KUKA KRL program: MyProgram_341().src

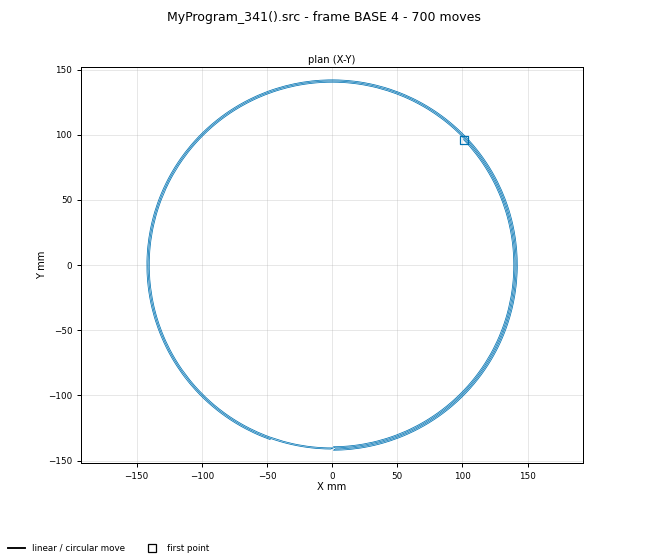
[picture p0: tool path of MyProgram_341().src in frame BASE 4, 700 of 700 moves have a stored position in this frame; points joined in program order, loops and branches not executed]
&ACCESS RVP
&REL 1
&PARAM TEMPLATE = C:\KRC\Roboter\Template\vorgabe
&PARAM EDITMASK = *
DEF MyProgram_341()
; ---- Setting reference (Base) ----
$BASE = BASE_DATA[4]

; --------------------------
; ---- Setting tool (TCP) ----
$TOOL = TOOL_DATA[3]
; --------------------------

$VEL.CP = VEL_APROX_PRINT
Startdeposition()
$VEL.CP = VEL_PRINT
LIN {X 100.8445,Y 96.2185,Z 191,A 42.0975,B 0.9774,C -0.019,E1 1.0995,E2 412.4998} C_DIS
LIN {X 103.8086,Y 93.0127,Z 191,A 40.4177,B 0.9774,C -0.0155,E1 1.1026,E2 414.1663} C_DIS
LIN {X 106.2355,Y 90.231,Z 191,A 38.3434,B 0.9775,C -0.0094,E1 1.1065,E2 416.3061} C_DIS
LIN {X 110.6605,Y 84.7459,Z 191,A 36.5482,B 0.9775,C -0.0077,E1 1.1094,E2 417.9718} C_DIS
LIN {X 113.1672,Y 81.369,Z 191,A 34.9648,B 0.9775,C -0.0043,E1 1.1119,E2 419.5381} C_DIS
LIN {X 115.7129,Y 77.7063,Z 191,A 33.5143,B 0.9775,C -0.0016,E1 1.1142,E2 420.9429} C_DIS
LIN {X 117.8631,Y 74.4035,Z 191,A 31.9484,B 0.9775,C 0.0021,E1 1.1165,E2 422.5025} C_DIS
LIN {X 120.2559,Y 70.4708,Z 191,A 30.262,B 0.9775,C 0.0059,E1 1.1189,E2 424.1645} C_DIS
LIN {X 122.5255,Y 66.4472,Z 191,A 28.5444,B 0.9775,C 0.0098,E1 1.1212,E2 425.8605} C_DIS
LIN {X 124.3166,Y 63.0275,Z 191,A 27.3294,B 0.9775,C 0.012,E1 1.1227,E2 427.0302} C_DIS
LIN {X 125.8319,Y 59.9448,Z 191,A 26.0722,B 0.9775,C 0.0149,E1 1.1242,E2 428.2687} C_DIS
LIN {X 128.0883,Y 54.9597,Z 191,A 23.995,B 0.9774,C 0.02,E1 1.1266,E2 430.3255} C_DIS
LIN {X 129.697,Y 51.0498,Z 191,A 22.4291,B 0.9774,C 0.0237,E1 1.1282,E2 431.8706} C_DIS
LIN {X 130.9681,Y 47.693,Z 191,A 21.1977,B 0.9772,C 0.0264,E1 1.1294,E2 433.0721} C_DIS
LIN {X 132.2016,Y 44.1567,Z 191,A 19.8499,B 0.9772,C 0.0295,E1 1.1306,E2 434.3965} C_DIS
LIN {X 133.196,Y 41.0607,Z 191,A 18.7703,B 0.9771,C 0.0318,E1 1.1314,E2 435.4443} C_DIS
LIN {X 134.1502,Y 37.8272,Z 191,A 17.3189,B 0.9769,C 0.0359,E1 1.1326,E2 436.9045} C_DIS
LIN {X 135.4414,Y 32.9058,Z 191,A 15.6224,B 0.9768,C 0.0396,E1 1.1337,E2 438.552} C_DIS
LIN {X 136.2147,Y 29.541,Z 191,A 14.3967,B 0.9767,C 0.0425,E1 1.1344,E2 439.7537} C_DIS
LIN {X 136.8872,Y 26.249,Z 191,A 12.5903,B 0.9764,C 0.0485,E1 1.1354,E2 441.6147} C_DIS
LIN {X 137.8072,Y 20.8924,Z 191,A 11.137,B 0.9763,C 0.0506,E1 1.136,E2 442.9697} C_DIS
LIN {X 138.3728,Y 16.7382,Z 191,A 9.6483,B 0.9761,C 0.0541,E1 1.1365,E2 444.4291} C_DIS
LIN {X 138.8051,Y 12.6771,Z 191,A 8.2382,B 0.9759,C 0.0574,E1 1.1369,E2 445.8054} C_DIS
LIN {X 139.1203,Y 8.5272,Z 191,A 6.7214,B 0.9757,C 0.0611,E1 1.1372,E2 447.2978} C_DIS
LIN {X 139.3137,Y 4.3756,Z 191,A 5.1532,B 0.9754,C 0.0651,E1 1.1374,E2 448.8488} C_DIS
LIN {X 139.3836,Y 0.2246,Z 191,A 3.614,B 0.9752,C 0.069,E1 1.1374,E2 450.3672} C_DIS
LIN {X 139.3302,Y -3.7808,Z 191,A 2.2878,B 0.9749,C 0.0719,E1 1.1374,E2 451.6522} C_DIS
LIN {X 139.1564,Y -7.9417,Z 191,A 0.7291,B 0.9746,C 0.0758,E1 1.1371,E2 453.1919} C_DIS
LIN {X 138.8913,Y -11.6781,Z 191,A -0.5528,B 0.9744,C 0.0787,E1 1.1368,E2 454.4406} C_DIS
LIN {X 138.519,Y -15.4917,Z 191,A -2.0184,B 0.9741,C 0.0825,E1 1.1364,E2 455.8927} C_DIS
LIN {X 138.008,Y -19.5189,Z 191,A -3.3769,B 0.9738,C 0.0855,E1 1.1359,E2 457.2109} C_DIS
LIN {X 137.3215,Y -23.8827,Z 191,A -5.0767,B 0.9735,C 0.0899,E1 1.1352,E2 458.8964} C_DIS
LIN {X 135.348,Y -33.2922,Z 191,A -8.6245,B 0.9726,C 0.0986,E1 1.1331,E2 462.3925} C_DIS
LIN {X 134.1503,Y -37.8269,Z 191,A -10.132,B 0.9723,C 0.1016,E1 1.132,E2 463.8445} C_DIS
LIN {X 133.1919,Y -41.0742,Z 191,A -11.393,B 0.972,C 0.1046,E1 1.131,E2 465.0888} C_DIS
LIN {X 132.027,Y -44.681,Z 191,A -12.8025,B 0.9716,C 0.108,E1 1.1298,E2 466.4792} C_DIS
LIN {X 130.6228,Y -48.6293,Z 191,A -14.2703,B 0.9712,C 0.1113,E1 1.1284,E2 467.9133} C_DIS
LIN {X 129.3401,Y -51.9444,Z 191,A -15.4509,B 0.971,C 0.1136,E1 1.1273,E2 469.0566} C_DIS
LIN {X 128.1203,Y -54.8857,Z 191,A -16.7235,B 0.9706,C 0.1169,E1 1.1259,E2 470.3252} C_DIS
LIN {X 126.5632,Y -58.385,Z 191,A -18.3527,B 0.97,C 0.1213,E1 1.124,E2 471.963} C_DIS
LIN {X 125.0675,Y -61.5237,Z 191,A -19.3037,B 0.9699,C 0.1225,E1 1.1229,E2 472.8492} C_DIS
LIN {X 123.5214,Y -64.5721,Z 191,A -20.5873,B 0.9695,C 0.1254,E1 1.1213,E2 474.117} C_DIS
LIN {X 121.4342,Y -68.4204,Z 191,A -22.2474,B 0.969,C 0.1292,E1 1.119,E2 475.7592} C_DIS
LIN {X 117.5792,Y -74.8523,Z 191,A -25.0092,B 0.9682,C 0.1352,E1 1.1151,E2 478.4787} C_DIS
LIN {X 115.0876,Y -78.629,Z 191,A -26.6462,B 0.9677,C 0.1386,E1 1.1126,E2 480.0859} C_DIS
LIN {X 112.552,Y -82.2179,Z 191,A -28.2704,B 0.9672,C 0.142,E1 1.11,E2 481.686} C_DIS
LIN {X 109.8372,Y -85.8109,Z 191,A -29.9359,B 0.9667,C 0.1454,E1 1.1072,E2 483.3268} C_DIS
LIN {X 106.958,Y -89.3737,Z 191,A -31.6211,B 0.9662,C 0.1488,E1 1.1042,E2 484.9856} C_DIS
LIN {X 104.0833,Y -92.706,Z 191,A -33.2121,B 0.9657,C 0.1518,E1 1.1013,E2 486.5471} C_DIS
LIN {X 101.0542,Y -95.9991,Z 191,A -34.8822,B 0.9652,C 0.1551,E1 1.0982,E2 488.1947} C_DIS
LIN {X 97.8841,Y -99.2293,Z 191,A -36.565,B 0.9647,C 0.1582,E1 1.0949,E2 489.8537} C_DIS
LIN {X 94.7472,Y -102.2285,Z 191,A -38.1412,B 0.9642,C 0.161,E1 1.0917,E2 491.4017} C_DIS
LIN {X 91.3868,Y -105.2433,Z 191,A -39.8212,B 0.9637,C 0.164,E1 1.0882,E2 493.0579} C_DIS
LIN {X 87.9612,Y -108.1227,Z 191,A -41.4803,B 0.9632,C 0.1669,E1 1.0847,E2 494.6926} C_DIS
LIN {X 84.472,Y -110.87,Z 191,A -43.1407,B 0.9628,C 0.1697,E1 1.081,E2 496.3307} C_DIS
LIN {X 80.7896,Y -113.5815,Z 191,A -44.8575,B 0.9623,C 0.1725,E1 1.0772,E2 498.0255} C_DIS
LIN {X 77.1218,Y -116.1031,Z 191,A -46.5386,B 0.9618,C 0.1752,E1 1.0733,E2 499.6865} C_DIS
LIN {X 73.2603,Y -118.5779,Z 191,A -48.3012,B 0.9613,C 0.178,E1 1.0691,E2 501.4329} C_DIS
LIN {X 69.8608,Y -120.6112,Z 191,A -49.8943,B 0.9608,C 0.1806,E1 1.0653,E2 503.0221} C_DIS
LIN {X 65.5664,Y -122.9992,Z 191,A -51.6426,B 0.9604,C 0.1828,E1 1.061,E2 504.7325} C_DIS
LIN {X 62.4534,Y -124.6089,Z 191,A -52.8854,B 0.9601,C 0.1842,E1 1.058,E2 505.9477} C_DIS
LIN {X 59.6812,Y -125.9579,Z 191,A -54.3785,B 0.9595,C 0.1871,E1 1.0541,E2 507.4745} C_DIS
LIN {X 56.1986,Y -127.5514,Z 191,A -55.6,B 0.9594,C 0.188,E1 1.0511,E2 508.6458} C_DIS
LIN {X 52.2827,Y -129.2037,Z 191,A -57.1304,B 0.959,C 0.1896,E1 1.0472,E2 510.1459} C_DIS
LIN {X 49.3407,Y -130.3564,Z 191,A -58.3976,B 0.9587,C 0.1912,E1 1.0439,E2 511.4093} C_DIS
LIN {X 45.7816,Y -131.6477,Z 191,A -59.8421,B 0.9584,C 0.1928,E1 1.0401,E2 512.8386} C_DIS
LIN {X 41.2319,Y -133.1436,Z 191,A -61.6603,B 0.958,C 0.1947,E1 1.0352,E2 514.6361} C_DIS
LIN {X 37.7566,Y -134.17,Z 191,A -62.9003,B 0.9579,C 0.1955,E1 1.032,E2 515.8404} C_DIS
LIN {X 34.7406,Y -134.983,Z 191,A -64.2072,B 0.9575,C 0.197,E1 1.0284,E2 517.1516} C_DIS
LIN {X 31.2504,Y -135.8329,Z 191,A -65.6672,B 0.9572,C 0.1985,E1 1.0244,E2 518.6101} C_DIS
LIN {X 24.229,Y -137.2596,Z 191,A -68.5094,B 0.9567,C 0.2009,E1 1.0165,E2 521.4391} C_DIS
LIN {X 19.9228,Y -137.9502,Z 191,A -70.2698,B 0.9564,C 0.2023,E1 1.0116,E2 523.1958} C_DIS
LIN {X 15.9492,Y -138.4669,Z 191,A -71.9027,B 0.9562,C 0.2036,E1 1.007,E2 524.8277} C_DIS
LIN {X 12.1677,Y -138.8499,Z 191,A -73.3225,B 0.956,C 0.2042,E1 1.0031,E2 526.2274} C_DIS
LIN {X 8.3965,Y -139.1284,Z 191,A -74.8296,B 0.9559,C 0.205,E1 0.9989,E2 527.7284} C_DIS
LIN {X 4.4323,Y -139.3121,Z 191,A -76.4575,B 0.9557,C 0.2059,E1 0.9943,E2 529.3567} C_DIS
LIN {X 0.9891,Y -139.3743,Z 191,A -77.3358,B 0.9559,C 0.205,E1 0.992,E2 530.156} C_DIS
Enddeposition()
LIN {X 0.9891,Y -139.3743,Z 191,A -77.3359,B 0.9559,C 0.205,E1 0.992,E2 530.1562} C_DIS
Startdeposition()
$VEL.CP = VEL_PRINT
LIN {X 2.4288,Y -140.2594,Z 191,A -76.5258,B 0.9476,C 0.2041,E1 0.9859,E2 529.3391} C_DIS
LIN {X 6.4097,Y -140.1353,Z 191,A -74.8363,B 0.9478,C 0.203,E1 0.9907,E2 527.6393} C_DIS
LIN {X 10.5728,Y -139.8818,Z 191,A -73.3277,B 0.9479,C 0.2025,E1 0.9949,E2 526.159} C_DIS
LIN {X 13.5665,Y -139.6228,Z 191,A -72.0791,B 0.9481,C 0.2016,E1 0.9984,E2 524.9064} C_DIS
LIN {X 17.8568,Y -139.1395,Z 191,A -70.3527,B 0.9484,C 0.2003,E1 1.0033,E2 523.1845} C_DIS
LIN {X 21.4621,Y -138.6287,Z 191,A -68.9845,B 0.9486,C 0.1995,E1 1.0071,E2 521.8332} C_DIS
LIN {X 24.5478,Y -138.1157,Z 191,A -67.4888,B 0.949,C 0.1976,E1 1.0113,E2 520.304} C_DIS
LIN {X 27.7783,Y -137.5024,Z 191,A -66.1559,B 0.9492,C 0.1963,E1 1.015,E2 518.9718} C_DIS
LIN {X 31.2997,Y -136.7437,Z 191,A -65.0397,B 0.9492,C 0.1961,E1 1.0179,E2 517.9078} C_DIS
LIN {X 34.4904,Y -135.9739,Z 191,A -63.7984,B 0.9495,C 0.195,E1 1.0213,E2 516.6805} C_DIS
LIN {X 38.0281,Y -135.0274,Z 191,A -62.3767,B 0.9498,C 0.1936,E1 1.0251,E2 515.2687} C_DIS
LIN {X 43.6634,Y -133.3133,Z 191,A -60.1874,B 0.9502,C 0.1915,E1 1.031,E2 513.1102} C_DIS
LIN {X 46.3959,Y -132.3862,Z 191,A -59.034,B 0.9505,C 0.1901,E1 1.034,E2 511.9596} C_DIS
LIN {X 49.306,Y -131.3293,Z 191,A -57.8285,B 0.9508,C 0.1886,E1 1.0372,E2 510.762} C_DIS
LIN {X 52.5839,Y -130.0515,Z 191,A -56.476,B 0.9511,C 0.187,E1 1.0407,E2 509.421} C_DIS
LIN {X 55.9899,Y -128.6222,Z 191,A -54.2348,B 0.9521,C 0.1817,E1 1.0468,E2 507.0695} C_DIS
LIN {X 62.3622,Y -125.6563,Z 191,A -52.699,B 0.9519,C 0.1829,E1 1.0502,E2 505.7302} C_DIS
LIN {X 64.8781,Y -124.376,Z 191,A -50.8289,B 0.9528,C 0.178,E1 1.0551,E2 503.7532} C_DIS
LIN {X 69.4356,Y -121.8922,Z 191,A -49.6152,B 0.9528,C 0.1784,E1 1.0578,E2 502.672} C_DIS
LIN {X 72.0547,Y -120.3627,Z 191,A -48.2313,B 0.9533,C 0.1756,E1 1.0612,E2 501.2658} C_DIS
LIN {X 75.8829,Y -117.9867,Z 191,A -46.4993,B 0.9538,C 0.1728,E1 1.0653,E2 499.5484} C_DIS
LIN {X 79.5681,Y -115.5334,Z 191,A -44.87,B 0.9542,C 0.1703,E1 1.069,E2 497.944} C_DIS
LIN {X 83.324,Y -112.8549,Z 191,A -43.1765,B 0.9547,C 0.1676,E1 1.0728,E2 496.277} C_DIS
LIN {X 86.9126,Y -110.1149,Z 191,A -41.4764,B 0.9552,C 0.1647,E1 1.0766,E2 494.5965} C_DIS
LIN {X 90.1823,Y -107.453,Z 191,A -39.9215,B 0.9557,C 0.162,E1 1.0799,E2 493.0647} C_DIS
LIN {X 93.5979,Y -104.4913,Z 191,A -38.2596,B 0.9562,C 0.1591,E1 1.0833,E2 491.4283} C_DIS
LIN {X 97.0336,Y -101.3089,Z 191,A -36.5299,B 0.9567,C 0.1559,E1 1.0868,E2 489.7237} C_DIS
LIN {X 100.354,Y -98.0212,Z 191,A -34.8379,B 0.9572,C 0.1528,E1 1.0901,E2 488.0616} C_DIS
LIN {X 103.4196,Y -94.781,Z 191,A -33.1724,B 0.9577,C 0.1495,E1 1.0932,E2 486.4173} C_DIS
LIN {X 106.4882,Y -91.32,Z 191,A -31.4671,B 0.9582,C 0.1462,E1 1.0963,E2 484.7371} C_DIS
LIN {X 109.4817,Y -87.7094,Z 191,A -29.754,B 0.9588,C 0.1427,E1 1.0993,E2 483.0516} C_DIS
LIN {X 112.2376,Y -84.1541,Z 191,A -28.1375,B 0.9592,C 0.1395,E1 1.102,E2 481.4654} C_DIS
LIN {X 114.7766,Y -80.656,Z 191,A -26.5389,B 0.9597,C 0.1362,E1 1.1046,E2 479.8893} C_DIS
LIN {X 117.2996,Y -76.9406,Z 191,A -24.9364,B 0.9602,C 0.1329,E1 1.107,E2 478.3184} C_DIS
LIN {X 120.1916,Y -72.3397,Z 191,A -22.7561,B 0.9609,C 0.1276,E1 1.1102,E2 476.1421} C_DIS
LIN {X 121.982,Y -69.2782,Z 191,A -21.7324,B 0.9611,C 0.1262,E1 1.1116,E2 475.1776} C_DIS
LIN {X 123.3706,Y -66.7748,Z 191,A -20.607,B 0.9614,C 0.1234,E1 1.1131,E2 474.0575} C_DIS
LIN {X 125.2761,Y -63.1242,Z 191,A -19.0934,B 0.9619,C 0.12,E1 1.1149,E2 472.5664} C_DIS
LIN {X 127.8258,Y -57.7868,Z 191,A -17.1962,B 0.9623,C 0.1165,E1 1.1171,E2 470.7403} C_DIS
LIN {X 129.5247,Y -53.8686,Z 191,A -15.5699,B 0.9628,C 0.1125,E1 1.1189,E2 469.1292} C_DIS
LIN {X 130.7911,Y -50.7163,Z 191,A -14.2895,B 0.9631,C 0.1094,E1 1.1202,E2 467.8627} C_DIS
LIN {X 132.3941,Y -46.373,Z 191,A -12.3171,B 0.9637,C 0.1039,E1 1.122,E2 465.8777} C_DIS
LIN {X 133.6698,Y -42.5544,Z 191,A -11.2361,B 0.9639,C 0.1025,E1 1.1229,E2 464.8738} C_DIS
LIN {X 134.773,Y -38.9229,Z 191,A -9.7971,B 0.9643,C 0.0989,E1 1.124,E2 463.4492} C_DIS
LIN {X 136.6408,Y -31.7502,Z 191,A -7.3212,B 0.9648,C 0.0937,E1 1.1257,E2 461.0471} C_DIS
LIN {X 137.2829,Y -28.8532,Z 191,A -6.168,B 0.9651,C 0.0906,E1 1.1264,E2 459.9012} C_DIS
LIN {X 137.9304,Y -25.5795,Z 191,A -4.8144,B 0.9654,C 0.0869,E1 1.1271,E2 458.548} C_DIS
LIN {X 138.7105,Y -20.9335,Z 191,A -3.3224,B 0.9657,C 0.084,E1 1.1277,E2 457.1136} C_DIS
LIN {X 139.1128,Y -18.0608,Z 191,A -2.2563,B 0.9659,C 0.0813,E1 1.1281,E2 456.0628} C_DIS
LIN {X 139.5316,Y -14.483,Z 191,A -0.9051,B 0.9662,C 0.0779,E1 1.1285,E2 454.7269} C_DIS
LIN {X 139.9067,Y -10.2319,Z 191,A 0.5882,B 0.9665,C 0.0744,E1 1.1288,E2 453.2663} C_DIS
LIN {X 140.1401,Y -6.3129,Z 191,A 1.9488,B 0.9667,C 0.0712,E1 1.129,E2 451.9374} C_DIS
LIN {X 140.2396,Y -3.4171,Z 191,A 3.1048,B 0.9669,C 0.068,E1 1.1291,E2 450.7843} C_DIS
LIN {X 140.2798,Y 0.701,Z 191,A 4.5452,B 0.9672,C 0.0646,E1 1.1291,E2 449.3754} C_DIS
LIN {X 140.1875,Y 5.1167,Z 191,A 6.0969,B 0.9674,C 0.061,E1 1.1291,E2 447.8562} C_DIS
LIN {X 140.0016,Y 8.8416,Z 191,A 7.3737,B 0.9676,C 0.058,E1 1.1288,E2 446.6112} C_DIS
LIN {X 139.7754,Y 11.8919,Z 191,A 8.4772,B 0.9677,C 0.0553,E1 1.1286,E2 445.5262} C_DIS
LIN {X 139.4287,Y 15.4394,Z 191,A 9.7987,B 0.9679,C 0.052,E1 1.1282,E2 444.2217} C_DIS
LIN {X 138.9585,Y 19.2214,Z 191,A 11.2418,B 0.9681,C 0.0483,E1 1.1277,E2 442.7928} C_DIS
LIN {X 138.162,Y 24.2893,Z 191,A 13.2764,B 0.9684,C 0.0428,E1 1.1267,E2 440.7651} C_DIS
LIN {X 137.4641,Y 27.9666,Z 191,A 14.449,B 0.9684,C 0.0405,E1 1.1261,E2 439.6384} C_DIS
LIN {X 136.328,Y 33.0638,Z 191,A 16.1697,B 0.9686,C 0.0368,E1 1.125,E2 437.9702} C_DIS
LIN {X 134.7053,Y 39.1541,Z 191,A 18.2378,B 0.9688,C 0.0324,E1 1.1236,E2 435.9662} C_DIS
LIN {X 133.5293,Y 42.9941,Z 191,A 19.8571,B 0.9689,C 0.0281,E1 1.1222,E2 434.3489} C_DIS
LIN {X 132.4144,Y 46.3145,Z 191,A 21.1201,B 0.9689,C 0.0251,E1 1.1211,E2 433.1068} C_DIS
LIN {X 131.2205,Y 49.5964,Z 191,A 22.3533,B 0.9691,C 0.0223,E1 1.1199,E2 431.8977} C_DIS
LIN {X 129.9725,Y 52.7799,Z 191,A 23.5651,B 0.9691,C 0.0195,E1 1.1187,E2 430.7088} C_DIS
LIN {X 128.8122,Y 55.5506,Z 191,A 24.8376,B 0.9691,C 0.0161,E1 1.1173,E2 429.4301} C_DIS
LIN {X 126.793,Y 60.0185,Z 191,A 26.3297,B 0.9692,C 0.0134,E1 1.1156,E2 428.0017} C_DIS
LIN {X 124.8732,Y 63.9155,Z 191,A 28.0232,B 0.9692,C 0.0092,E1 1.1135,E2 426.3178} C_DIS
LIN {X 123.0071,Y 67.4414,Z 191,A 29.5422,B 0.9693,C 0.0056,E1 1.1115,E2 424.8122} C_DIS
LIN {X 120.7502,Y 71.4042,Z 191,A 31.1652,B 0.9693,C 0.0021,E1 1.1093,E2 423.2186} C_DIS
LIN {X 118.4379,Y 75.177,Z 191,A 33.1475,B 0.9693,C -0.0032,E1 1.1063,E2 421.2142} C_DIS
LIN {X 115.92,Y 79.0046,Z 191,A 34.5042,B 0.9693,C -0.0053,E1 1.1043,E2 419.9209} C_DIS
LIN {X 113.0722,Y 83.0281,Z 191,A 36.2138,B 0.9693,C -0.0087,E1 1.1015,E2 418.2482} C_DIS
LIN {X 110.078,Y 86.9578,Z 191,A 38.2225,B 0.9693,C -0.0134,E1 1.098,E2 416.2402} C_DIS
LIN {X 107.8514,Y 89.7059,Z 191,A 39.2586,B 0.9693,C -0.0149,E1 1.0963,E2 415.2538} C_DIS
LIN {X 105.0814,Y 92.9348,Z 191,A 40.865,B 0.9691,C -0.0182,E1 1.0934,E2 413.663} C_DIS
LIN {X 101.9188,Y 96.3928,Z 191,A 42.5668,B 0.9691,C -0.0215,E1 1.0902,E2 411.9867} C_DIS
LIN {X 98.7421,Y 99.6445,Z 191,A 44.3488,B 0.969,C -0.0253,E1 1.0866,E2 410.2135} C_DIS
LIN {X 93.6427,Y 104.4511,Z 191,A 46.6153,B 0.9689,C -0.0287,E1 1.0821,E2 408.0181} C_DIS
LIN {X 91.2896,Y 106.5144,Z 191,A 47.9945,B 0.9688,C -0.0318,E1 1.0792,E2 406.6268} C_DIS
LIN {X 87.7142,Y 109.4778,Z 191,A 49.6935,B 0.9687,C -0.0348,E1 1.0755,E2 404.9513} C_DIS
LIN {X 84.1709,Y 112.2249,Z 191,A 51.39,B 0.9686,C -0.0378,E1 1.0718,E2 403.2707} C_DIS
LIN {X 78.7346,Y 116.1028,Z 191,A 53.9921,B 0.9684,C -0.0424,E1 1.0658,E2 400.6835} C_DIS
LIN {X 74.2059,Y 119.0483,Z 191,A 55.875,B 0.9683,C -0.0451,E1 1.0614,E2 398.8387} C_DIS
LIN {X 70.7179,Y 121.1533,Z 191,A 57.4143,B 0.9682,C -0.0475,E1 1.0577,E2 397.314} C_DIS
LIN {X 66.6844,Y 123.4192,Z 191,A 59.1449,B 0.968,C -0.05,E1 1.0535,E2 395.6021} C_DIS
LIN {X 62.523,Y 125.5769,Z 191,A 60.8209,B 0.968,C -0.0522,E1 1.0493,E2 393.9539} C_DIS
LIN {X 58.5898,Y 127.4589,Z 191,A 62.4897,B 0.9678,C -0.0545,E1 1.0451,E2 392.2982} C_DIS
LIN {X 55.4025,Y 128.8762,Z 191,A 63.7787,B 0.9677,C -0.0561,E1 1.0418,E2 391.0251} C_DIS
LIN {X 51.8629,Y 130.3421,Z 191,A 65.2128,B 0.9676,C -0.0579,E1 1.0381,E2 389.6062} C_DIS
LIN {X 48.9366,Y 131.4676,Z 191,A 66.4229,B 0.9675,C -0.0594,E1 1.0349,E2 388.4044} C_DIS
LIN {X 45.7519,Y 132.6095,Z 191,A 67.7199,B 0.9675,C -0.0609,E1 1.0315,E2 387.1173} C_DIS
LIN {X 42.6175,Y 133.6496,Z 191,A 70.0962,B 0.9671,C -0.0659,E1 1.0248,E2 384.6231} C_DIS
LIN {X 34.6875,Y 135.9239,Z 191,A 71.9236,B 0.9671,C -0.0648,E1 1.0203,E2 382.9733} C_DIS
LIN {X 30.496,Y 136.9262,Z 191,A 74.095,B 0.9669,C -0.068,E1 1.0142,E2 380.7559} C_DIS
LIN {X 27.1654,Y 137.6271,Z 191,A 75.1328,B 0.9669,C -0.0683,E1 1.0114,E2 379.7584} C_DIS
LIN {X 24.2811,Y 138.1634,Z 191,A 76.3446,B 0.9669,C -0.0694,E1 1.008,E2 378.5453} C_DIS
LIN {X 19.9734,Y 138.8511,Z 191,A 78.0673,B 0.9667,C -0.0708,E1 1.0033,E2 376.8298} C_DIS
LIN {X 16.0453,Y 139.3608,Z 191,A 79.5373,B 0.9667,C -0.0716,E1 0.9992,E2 375.377} C_DIS
LIN {X 11.9143,Y 139.7735,Z 191,A 81.1822,B 0.9666,C -0.0727,E1 0.9946,E2 373.7383} C_DIS
LIN {X 8.3688,Y 140.0307,Z 191,A 82.5796,B 0.9666,C -0.0734,E1 0.9906,E2 372.3475} C_DIS
LIN {X 4.3944,Y 140.2124,Z 191,A 84.238,B 0.9665,C -0.0744,E1 0.9859,E2 370.686} C_DIS
LIN {X 0.4701,Y 140.28,Z 191,A 85.7526,B 0.9665,C -0.075,E1 0.9817,E2 369.1818} C_DIS
LIN {X -3.8447,Y 140.2277,Z 191,A 87.4841,B 0.9664,C -0.0756,E1 0.9768,E2 367.4543} C_DIS
LIN {X -8.1948,Y 140.0414,Z 191,A 89.2607,B 0.9664,C -0.0762,E1 0.9718,E2 365.6787} C_DIS
LIN {X -11.8972,Y 139.7749,Z 191,A 90.7411,B 0.9664,C -0.0765,E1 0.9676,E2 364.2029} C_DIS
LIN {X -16.0691,Y 139.3579,Z 191,A 92.4601,B 0.9663,C -0.0767,E1 0.9628,E2 362.4839} C_DIS
LIN {X -20.8516,Y 138.7232,Z 191,A 94.5728,B 0.9663,C -0.0771,E1 0.9568,E2 360.3563} C_DIS
LIN {X -24.7655,Y 138.0768,Z 191,A 95.986,B 0.9663,C -0.0767,E1 0.9529,E2 358.9668} C_DIS
LIN {X -28.6695,Y 137.3211,Z 191,A 97.6024,B 0.9663,C -0.0765,E1 0.9484,E2 357.3521} C_DIS
LIN {X -32.3615,Y 136.4972,Z 191,A 99.0478,B 0.9663,C -0.0761,E1 0.9445,E2 355.9184} C_DIS
LIN {X -35.0189,Y 135.8398,Z 191,A 100.2628,B 0.9663,C -0.076,E1 0.9411,E2 354.6932} C_DIS
LIN {X -37.9053,Y 135.0618,Z 191,A 101.5938,B 0.9663,C -0.0758,E1 0.9375,E2 353.3506} C_DIS
LIN {X -41.2345,Y 134.0829,Z 191,A 103.0152,B 0.9663,C -0.0753,E1 0.9336,E2 351.9294} C_DIS
LIN {X -44.7517,Y 132.9509,Z 191,A 104.5488,B 0.9664,C -0.0746,E1 0.9295,E2 350.3939} C_DIS
LIN {X -48.4055,Y 131.6665,Z 191,A 106.1601,B 0.9665,C -0.0739,E1 0.9252,E2 348.7802} C_DIS
LIN {X -51.1258,Y 130.6319,Z 191,A 107.4182,B 0.9665,C -0.0732,E1 0.9218,E2 347.5149} C_DIS
LIN {X -56.4675,Y 128.4137,Z 191,A 109.9431,B 0.9667,C -0.0718,E1 0.9152,E2 344.9731} C_DIS
LIN {X -59.2165,Y 127.1691,Z 191,A 111.1417,B 0.9667,C -0.0708,E1 0.9122,E2 343.7789} C_DIS
LIN {X -62.702,Y 125.4886,Z 191,A 112.7735,B 0.9668,C -0.0696,E1 0.908,E2 342.1423} C_DIS
LIN {X -65.7052,Y 123.9417,Z 191,A 114.2628,B 0.9669,C -0.0684,E1 0.9042,E2 340.6415} C_DIS
LIN {X -70.5272,Y 121.2641,Z 191,A 116.7091,B 0.967,C -0.0663,E1 0.8982,E2 338.1747} C_DIS
LIN {X -74.6394,Y 118.7772,Z 191,A 118.7378,B 0.9672,C -0.0642,E1 0.8933,E2 336.1397} C_DIS
LIN {X -78.1585,Y 116.4918,Z 191,A 120.775,B 0.9673,C -0.0623,E1 0.8884,E2 334.0669} C_DIS
LIN {X -82.3299,Y 113.5816,Z 191,A 122.6839,B 0.9675,C -0.0596,E1 0.884,E2 332.1783} C_DIS
LIN {X -85.1351,Y 111.4945,Z 191,A 124.4137,B 0.9675,C -0.0578,E1 0.8801,E2 330.4151} C_DIS
LIN {X -88.798,Y 108.5997,Z 191,A 126.447,B 0.9678,C -0.0551,E1 0.8756,E2 328.3684} C_DIS
LIN {X -92.093,Y 105.8202,Z 191,A 128.4084,B 0.9679,C -0.0524,E1 0.8713,E2 326.385} C_DIS
LIN {X -95.4496,Y 102.8027,Z 191,A 130.4234,B 0.9681,C -0.0495,E1 0.8671,E2 324.3515} C_DIS
LIN {X -98.6352,Y 99.7507,Z 191,A 132.4213,B 0.9682,C -0.0465,E1 0.863,E2 322.332} C_DIS
LIN {X -101.8138,Y 96.5042,Z 191,A 134.4577,B 0.9684,C -0.0432,E1 0.859,E2 320.2757} C_DIS
LIN {X -104.8181,Y 93.2328,Z 191,A 136.4679,B 0.9685,C -0.0398,E1 0.8552,E2 318.2438} C_DIS
LIN {X -107.7692,Y 89.8052,Z 191,A 138.4956,B 0.9686,C -0.0362,E1 0.8515,E2 316.1961} C_DIS
LIN {X -110.5694,Y 86.3341,Z 191,A 140.6663,B 0.9688,C -0.0325,E1 0.8476,E2 313.9854} C_DIS
LIN {X -114.8976,Y 80.4844,Z 191,A 144.4492,B 0.969,C -0.026,E1 0.8413,E2 310.1078} C_DIS
LIN {X -117.6144,Y 76.4582,Z 191,A 146.1159,B 0.969,C -0.0219,E1 0.8387,E2 308.4803} C_DIS
LIN {X -121.8922,Y 69.4356,Z 191,A 149.6168,B 0.9692,C -0.0142,E1 0.8337,E2 304.9647} C_DIS
LIN {X -123.3498,Y 66.8131,Z 191,A 151.4066,B 0.9692,C -0.011,E1 0.8311,E2 303.1077} C_DIS
LIN {X -125.0943,Y 63.4813,Z 191,A 152.9992,B 0.9692,C -0.0073,E1 0.8291,E2 301.5092} C_DIS
LIN {X -127.4467,Y 58.6161,Z 191,A 155.444,B 0.9693,C -0.0018,E1 0.8261,E2 299.0369} C_DIS
LIN {X -129.9834,Y 52.753,Z 191,A 158.4922,B 0.9693,C 0.005,E1 0.8227,E2 295.9367} C_DIS
LIN {X -130.907,Y 50.4182,Z 191,A 159.7153,B 0.9693,C 0.0078,E1 0.8214,E2 294.6899} C_DIS
LIN {X -131.9573,Y 47.5997,Z 191,A 161.2886,B 0.9693,C 0.0112,E1 0.8199,E2 293.0746} C_DIS
LIN {X -133.199,Y 44.0068,Z 191,A 162.9736,B 0.9692,C 0.0153,E1 0.8184,E2 291.374} C_DIS
LIN {X -134.211,Y 40.816,Z 191,A 164.6066,B 0.9692,C 0.0191,E1 0.817,E2 289.7086} C_DIS
LIN {X -135.1979,Y 37.4185,Z 191,A 166.8546,B 0.969,C 0.0237,E1 0.8153,E2 287.3601} C_DIS
LIN {X -136.3308,Y 33.0521,Z 191,A 168.4865,B 0.969,C 0.0284,E1 0.8142,E2 285.7561} C_DIS
LIN {X -137.0064,Y 30.1337,Z 191,A 169.9402,B 0.9688,C 0.0319,E1 0.8133,E2 284.274} C_DIS
LIN {X -137.8444,Y 26.0295,Z 191,A 171.8674,B 0.9686,C 0.0368,E1 0.8122,E2 282.3202} C_DIS
LIN {X -139.0055,Y 18.8799,Z 191,A 175.8108,B 0.9682,C 0.0459,E1 0.8105,E2 278.2514} C_DIS
LIN {X -139.4832,Y 14.9325,Z 191,A 177.2484,B 0.968,C 0.0502,E1 0.8101,E2 276.839} C_DIS
LIN {X -139.8778,Y 10.6278,Z 191,A -179.6827,B 0.9677,C 0.0563,E1 0.8094,E2 273.6001} C_DIS
LIN {X -140.2195,Y 4.1391,Z 191,A -177.8678,B 0.9673,C 0.063,E1 0.8092,E2 271.8975} C_DIS
LIN {X -140.2443,Y -3.2474,Z 191,A -174.1217,B 0.9666,C 0.0721,E1 0.8092,E2 268.0572} C_DIS
LIN {X -139.8415,Y -11.1088,Z 191,A -170.0509,B 0.9659,C 0.0818,E1 0.8099,E2 263.874} C_DIS
LIN {X -139.2722,Y -16.7876,Z 191,A -167.5021,B 0.9653,C 0.0884,E1 0.8107,E2 261.2971} C_DIS
LIN {X -137.9392,Y -25.5336,Z 191,A -163.3295,B 0.9643,C 0.0988,E1 0.8126,E2 257.0506} C_DIS
LIN {X -137.3992,Y -28.2855,Z 191,A -161.9601,B 0.9639,C 0.102,E1 0.8133,E2 255.6511} C_DIS
LIN {X -136.7276,Y -31.3699,Z 191,A -160.4707,B 0.9635,C 0.1056,E1 0.8143,E2 254.1348} C_DIS
LIN {X -135.9581,Y -34.5525,Z 191,A -158.866,B 0.9631,C 0.1094,E1 0.8154,E2 252.4939} C_DIS
LIN {X -135.0462,Y -37.9609,Z 191,A -157.1666,B 0.9627,C 0.1134,E1 0.8166,E2 250.7594} C_DIS
LIN {X -134.0581,Y -41.3155,Z 191,A -155.5401,B 0.9622,C 0.1172,E1 0.818,E2 249.1061} C_DIS
LIN {X -132.6865,Y -45.5296,Z 191,A -152.9972,B 0.9616,C 0.1223,E1 0.8204,E2 246.4615} C_DIS
LIN {X -131.3592,Y -49.2262,Z 191,A -151.9914,B 0.9611,C 0.1261,E1 0.8213,E2 245.5401} C_DIS
LIN {X -130.6363,Y -51.1145,Z 191,A -150.635,B 0.9608,C 0.1284,E1 0.8227,E2 244.1098} C_DIS
LIN {X -128.913,Y -55.3174,Z 191,A -148.6681,B 0.9601,C 0.1331,E1 0.8248,E2 242.128} C_DIS
LIN {X -127.5583,Y -58.3749,Z 191,A -146.7657,B 0.9596,C 0.1366,E1 0.8271,E2 240.1503} C_DIS
LIN {X -125.7295,Y -62.2136,Z 191,A -145.0019,B 0.959,C 0.1408,E1 0.8293,E2 238.3832} C_DIS
LIN {X -124.3202,Y -64.9844,Z 191,A -143.5199,B 0.9586,C 0.1438,E1 0.8312,E2 236.8714} C_DIS
LIN {X -122.3736,Y -68.5838,Z 191,A -141.4833,B 0.958,C 0.1478,E1 0.834,E2 234.7832} C_DIS
LIN {X -120.1597,Y -72.3927,Z 191,A -139.3765,B 0.9574,C 0.1518,E1 0.8371,E2 232.6328} C_DIS
LIN {X -117.5681,Y -76.5295,Z 191,A -137.2553,B 0.9567,C 0.1562,E1 0.8403,E2 230.4938} C_DIS
LIN {X -115.1138,Y -80.1736,Z 191,A -135.1918,B 0.956,C 0.16,E1 0.8437,E2 228.3919} C_DIS
LIN {X -109.0235,Y -88.2776,Z 191,A -130.9065,B 0.9546,C 0.1683,E1 0.851,E2 224.0868} C_DIS
LIN {X -105.3142,Y -92.6716,Z 191,A -127.9292,B 0.9539,C 0.1725,E1 0.8566,E2 221.0184} C_DIS
LIN {X -102.2596,Y -96.0316,Z 191,A -125.8675,B 0.9533,C 0.1757,E1 0.8606,E2 218.9266} C_DIS
LIN {X -97.1105,Y -101.2354,Z 191,A -122.0719,B 0.9524,C 0.1802,E1 0.8685,E2 215.0126} C_DIS
LIN {X -93.4502,Y -104.6235,Z 191,A -120.0576,B 0.9518,C 0.1834,E1 0.8727,E2 213.0017} C_DIS
LIN {X -90.4494,Y -107.2288,Z 191,A -118.9223,B 0.9513,C 0.1862,E1 0.875,E2 211.9384} C_DIS
LIN {X -86.5162,Y -110.4263,Z 191,A -116.4374,B 0.9508,C 0.1888,E1 0.8806,E2 209.3923} C_DIS
LIN {X -82.1503,Y -113.7118,Z 191,A -114.075,B 0.9502,C 0.1916,E1 0.886,E2 207.0104} C_DIS
LIN {X -78.6984,Y -116.1273,Z 191,A -112.1661,B 0.9498,C 0.1934,E1 0.8905,E2 205.0735} C_DIS
LIN {X -75.1214,Y -118.473,Z 191,A -110.2949,B 0.9495,C 0.1953,E1 0.895,E2 203.1837} C_DIS
LIN {X -71.254,Y -120.8384,Z 191,A -108.3133,B 0.9491,C 0.197,E1 0.8998,E2 201.1824} C_DIS
LIN {X -67.1186,Y -123.1832,Z 191,A -106.1291,B 0.9488,C 0.1985,E1 0.9053,E2 198.9617} C_DIS
LIN {X -63.0139,Y -125.3322,Z 191,A -104.4884,B 0.9484,C 0.2005,E1 0.9093,E2 197.3582} C_DIS
LIN {X -60.216,Y -126.6986,Z 191,A -103.0657,B 0.9482,C 0.2013,E1 0.913,E2 195.9126} C_DIS
LIN {X -57.0526,Y -128.1542,Z 191,A -101.6196,B 0.948,C 0.2023,E1 0.9167,E2 194.4627} C_DIS
LIN {X -53.778,Y -129.5626,Z 191,A -100.1387,B 0.9478,C 0.2032,E1 0.9206,E2 192.9777} C_DIS
LIN {X -50.83,Y -130.7469,Z 191,A -98.752,B 0.9477,C 0.2038,E1 0.9243,E2 191.5772} C_DIS
LIN {X -47.4936,Y -131.9956,Z 191,A -97.257,B 0.9475,C 0.2045,E1 0.9283,E2 190.0758} C_DIS
LIN {X -37.0814,Y -135.2922,Z 191,A -92.7922,B 0.9471,C 0.2062,E1 0.9404,E2 185.6095} C_DIS
LIN {X -30.0812,Y -137.0177,Z 191,A -89.8663,B 0.9471,C 0.2068,E1 0.9484,E2 182.6853} C_DIS
LIN {X -26.3218,Y -137.7885,Z 191,A -88.1757,B 0.9471,C 0.2066,E1 0.9532,E2 180.9756} C_DIS
LIN {X -22.8732,Y -138.403,Z 191,A -86.7287,B 0.9471,C 0.2066,E1 0.9572,E2 179.5255} C_DIS
LIN {X -19.4647,Y -138.9238,Z 191,A -85.3227,B 0.9471,C 0.2065,E1 0.9611,E2 178.1193} C_DIS
LIN {X -15.7103,Y -139.3995,Z 191,A -83.6759,B 0.9471,C 0.206,E1 0.9658,E2 176.4566} C_DIS
LIN {X -11.1977,Y -139.834,Z 191,A -81.8256,B 0.9473,C 0.2056,E1 0.971,E2 174.6056} C_DIS
LIN {X -7.0178,Y -140.1047,Z 191,A -80.2259,B 0.9473,C 0.2054,E1 0.9755,E2 173.0218} C_DIS
LIN {X -3.4723,Y -140.238,Z 191,A -78.8632,B 0.9473,C 0.2051,E1 0.9793,E2 171.6713} C_DIS
LIN {X 0.9989,Y -140.2749,Z 191,A -77.1882,B 0.9475,C 0.2047,E1 0.984,E2 170.0179} C_DIS
Enddeposition()
LIN {X 0.9989,Y -140.2749,Z 191,A -77.1882,B 0.9475,C 0.2047,E1 0.984,E2 170.0179} C_DIS
Startdeposition()
$VEL.CP = VEL_PRINT
LIN {X -1.0513,Y -141.1757,Z 191,A -78.2711,B 0.9179,C 0.2049,E1 0.9515,E2 171.1715} C_DIS
LIN {X -5.3673,Y -141.0773,Z 191,A -79.9095,B 0.9179,C 0.2053,E1 0.9469,E2 172.7937} C_DIS
LIN {X -8.8162,Y -140.9038,Z 191,A -81.251,B 0.9178,C 0.2055,E1 0.9431,E2 174.1269} C_DIS
LIN {X -11.9765,Y -140.6703,Z 191,A -82.6035,B 0.9176,C 0.2061,E1 0.9393,E2 175.49} C_DIS
LIN {X -15.6835,Y -140.3065,Z 191,A -84.1899,B 0.9176,C 0.2065,E1 0.9348,E2 177.0884} C_DIS
LIN {X -19.9252,Y -139.766,Z 191,A -85.8094,B 0.9176,C 0.2065,E1 0.9303,E2 178.6912} C_DIS
LIN {X -23.2557,Y -139.2505,Z 191,A -87.1888,B 0.9176,C 0.2065,E1 0.9264,E2 180.073} C_DIS
LIN {X -26.8832,Y -138.5964,Z 191,A -88.6783,B 0.9176,C 0.2065,E1 0.9223,E2 181.5622} C_DIS
LIN {X -31.0404,Y -137.725,Z 191,A -90.8437,B 0.9174,C 0.2072,E1 0.9161,E2 183.7947} C_DIS
LIN {X -35.2441,Y -136.71,Z 191,A -92.1868,B 0.9177,C 0.206,E1 0.9126,E2 185.0766} C_DIS
LIN {X -39.285,Y -135.6036,Z 191,A -94.4882,B 0.9175,C 0.2067,E1 0.9061,E2 187.4688} C_DIS
LIN {X -44.1423,Y -134.1013,Z 191,A -96.1549,B 0.9179,C 0.2051,E1 0.9017,E2 189.0768} C_DIS
LIN {X -47.6713,Y -132.887,Z 191,A -97.5862,B 0.918,C 0.2043,E1 0.8979,E2 190.4959} C_DIS
LIN {X -51.201,Y -131.5672,Z 191,A -99.1565,B 0.9182,C 0.2035,E1 0.8938,E2 192.0729} C_DIS
LIN {X -54.692,Y -130.155,Z 191,A -100.7423,B 0.9184,C 0.2027,E1 0.8896,E2 193.6678} C_DIS
LIN {X -58.558,Y -128.464,Z 191,A -102.5916,B 0.9186,C 0.2017,E1 0.8848,E2 195.538} C_DIS
LIN {X -62.73,Y -126.4772,Z 191,A -104.491,B 0.9189,C 0.2003,E1 0.8799,E2 197.4413} C_DIS
LIN {X -67.6372,Y -123.9243,Z 191,A -106.9008,B 0.9193,C 0.1985,E1 0.8738,E2 199.8763} C_DIS
LIN {X -71.4441,Y -121.7693,Z 191,A -108.7794,B 0.9196,C 0.1969,E1 0.8692,E2 201.7706} C_DIS
LIN {X -75.3483,Y -119.3928,Z 191,A -110.7404,B 0.92,C 0.1951,E1 0.8644,E2 203.7477} C_DIS
LIN {X -79.286,Y -116.8151,Z 191,A -112.9014,B 0.9205,C 0.1931,E1 0.8593,E2 205.9461} C_DIS
LIN {X -85.4007,Y -112.423,Z 191,A -116.0931,B 0.9212,C 0.1893,E1 0.8519,E2 209.1583} C_DIS
LIN {X -89.0391,Y -109.5637,Z 191,A -118.1076,B 0.9217,C 0.1868,E1 0.8475,E2 211.193} C_DIS
LIN {X -93.133,Y -106.1057,Z 191,A -120.4873,B 0.9224,C 0.1838,E1 0.8423,E2 213.603} C_DIS
LIN {X -96.5044,Y -103.0488,Z 191,A -123.3072,B 0.9228,C 0.1814,E1 0.8362,E2 216.5654} C_DIS
LIN {X -101.0981,Y -98.5462,Z 191,A -125.0656,B 0.9238,C 0.1766,E1 0.833,E2 218.1991} C_DIS
LIN {X -104.341,Y -95.1055,Z 191,A -127.5123,B 0.9244,C 0.1734,E1 0.8281,E2 220.723} C_DIS
LIN {X -108.3032,Y -90.5675,Z 191,A -130.1894,B 0.9252,C 0.1689,E1 0.8231,E2 223.4336} C_DIS
LIN {X -114.419,Y -82.7063,Z 191,A -134.4476,B 0.9266,C 0.1609,E1 0.8158,E2 227.7227} C_DIS
LIN {X -116.1948,Y -80.1929,Z 191,A -136.1485,B 0.9271,C 0.1583,E1 0.8129,E2 229.4887} C_DIS
LIN {X -118.4424,Y -76.8336,Z 191,A -138.0895,B 0.9277,C 0.1548,E1 0.8099,E2 231.4727} C_DIS
LIN {X -121.0046,Y -72.7326,Z 191,A -140.2526,B 0.9284,C 0.1504,E1 0.8066,E2 233.664} C_DIS
LIN {X -123.2553,Y -68.8497,Z 191,A -142.288,B 0.9291,C 0.1462,E1 0.8038,E2 235.7295} C_DIS
LIN {X -125.2691,Y -65.1109,Z 191,A -144.183,B 0.9297,C 0.1422,E1 0.8013,E2 237.6483} C_DIS
LIN {X -126.8545,Y -61.9651,Z 191,A -145.81,B 0.9302,C 0.1387,E1 0.7992,E2 239.3029} C_DIS
LIN {X -128.1247,Y -59.2916,Z 191,A -147.2133,B 0.9306,C 0.1357,E1 0.7975,E2 240.7345} C_DIS
LIN {X -130.3082,Y -54.3252,Z 191,A -149.3643,B 0.9314,C 0.1304,E1 0.7951,E2 242.8776} C_DIS
LIN {X -131.0134,Y -52.6022,Z 191,A -150.6817,B 0.9317,C 0.1282,E1 0.7936,E2 244.2739} C_DIS
LIN {X -132.4704,Y -48.8223,Z 191,A -152.5168,B 0.9323,C 0.1239,E1 0.7918,E2 246.1351} C_DIS
LIN {X -134.1414,Y -44.0219,Z 191,A -154.9093,B 0.933,C 0.1184,E1 0.7896,E2 248.5728} C_DIS
LIN {X -135.064,Y -41.1003,Z 191,A -156.4027,B 0.9334,C 0.115,E1 0.7883,E2 250.1003} C_DIS
LIN {X -136.1666,Y -37.2922,Z 191,A -158.2728,B 0.934,C 0.1106,E1 0.7868,E2 252.006} C_DIS
LIN {X -136.8534,Y -34.6793,Z 191,A -159.5921,B 0.9343,C 0.1075,E1 0.7859,E2 253.3554} C_DIS
LIN {X -137.6691,Y -31.2851,Z 191,A -161.2482,B 0.9348,C 0.1035,E1 0.7848,E2 255.0437} C_DIS
LIN {X -138.4118,Y -27.8174,Z 191,A -162.9876,B 0.9352,C 0.0994,E1 0.7838,E2 256.8234} C_DIS
LIN {X -139.5224,Y -21.565,Z 191,A -165.9763,B 0.936,C 0.092,E1 0.7824,E2 259.8667} C_DIS
LIN {X -140.0381,Y -17.9182,Z 191,A -167.6938,B 0.9364,C 0.0877,E1 0.7817,E2 261.6136} C_DIS
LIN {X -140.8038,Y -10.2888,Z 191,A -171.9123,B 0.9373,C 0.078,E1 0.7806,E2 265.9783} C_DIS
LIN {X -141.0509,Y -6.0435,Z 191,A -173.2829,B 0.9376,C 0.0735,E1 0.7805,E2 267.3009} C_DIS
LIN {X -141.1721,Y -1.61,Z 191,A -176.1206,B 0.9381,C 0.0675,E1 0.7803,E2 270.2744} C_DIS
LIN {X -141.1546,Y 2.6634,Z 191,A -177.7312,B 0.9384,C 0.0627,E1 0.7803,E2 271.8679} C_DIS
LIN {X -140.8769,Y 9.2517,Z 191,A 179.3878,B 0.9389,C 0.0551,E1 0.7808,E2 274.7741} C_DIS
LIN {X -140.649,Y 12.229,Z 191,A 177.6771,B 0.9391,C 0.0512,E1 0.7812,E2 276.5489} C_DIS
LIN {X -140.2201,Y 16.4309,Z 191,A 175.6176,B 0.9394,C 0.0461,E1 0.7818,E2 278.6518} C_DIS
LIN {X -139.6199,Y 20.9318,Z 191,A 173.1853,B 0.9396,C 0.0404,E1 0.7828,E2 281.1583} C_DIS
LIN {X -139.0316,Y 24.533,Z 191,A 172.0931,B 0.9398,C 0.0368,E1 0.7833,E2 282.2001} C_DIS
LIN {X -137.6624,Y 31.3142,Z 191,A 168.8849,B 0.9401,C 0.0287,E1 0.7851,E2 285.4577} C_DIS
LIN {X -136.5886,Y 35.7144,Z 191,A 166.3485,B 0.9402,C 0.0231,E1 0.7869,E2 288.081} C_DIS
LIN {X -135.7771,Y 38.6852,Z 191,A 164.9063,B 0.9402,C 0.0196,E1 0.788,E2 289.5465} C_DIS
LIN {X -134.5861,Y 42.64,Z 191,A 162.9587,B 0.9404,C 0.015,E1 0.7896,E2 291.5267} C_DIS
LIN {X -133.1596,Y 46.9093,Z 191,A 160.8323,B 0.9404,C 0.01,E1 0.7916,E2 293.689} C_DIS
LIN {X -131.9126,Y 50.3115,Z 191,A 159.1442,B 0.9404,C 0.006,E1 0.7933,E2 295.4029} C_DIS
LIN {X -130.8668,Y 52.9657,Z 191,A 157.5885,B 0.9404,C 0.0028,E1 0.7949,E2 297.0064} C_DIS
LIN {X -129.0456,Y 57.2612,Z 191,A 155.4023,B 0.9404,C -0.0021,E1 0.7974,E2 299.2269} C_DIS
LIN {X -126.6937,Y 62.291,Z 191,A 153.2866,B 0.9404,C -0.0075,E1 0.7999,E2 301.3245} C_DIS
LIN {X -125.5932,Y 64.4827,Z 191,A 151.7061,B 0.9404,C -0.0103,E1 0.802,E2 302.975} C_DIS
LIN {X -123.2794,Y 68.8067,Z 191,A 148.8203,B 0.9404,C -0.0154,E1 0.8061,E2 305.9657} C_DIS
LIN {X -120.624,Y 73.362,Z 191,A 147.2806,B 0.9403,C -0.0199,E1 0.8082,E2 307.4333} C_DIS
LIN {X -118.8328,Y 76.2286,Z 191,A 145.4526,B 0.9403,C -0.0232,E1 0.811,E2 309.3143} C_DIS
LIN {X -115.7964,Y 80.7665,Z 191,A 143.0311,B 0.9401,C -0.0281,E1 0.8149,E2 311.7586} C_DIS
LIN {X -111.9259,Y 86.0507,Z 191,A 140.2392,B 0.9399,C -0.0336,E1 0.8196,E2 314.5645} C_DIS
LIN {X -108.8219,Y 89.9434,Z 191,A 137.6663,B 0.9397,C -0.0377,E1 0.8242,E2 317.2004} C_DIS
LIN {X -105.9763,Y 93.2798,Z 191,A 135.6478,B 0.9396,C -0.0411,E1 0.828,E2 319.2453} C_DIS
LIN {X -102.9039,Y 96.6586,Z 191,A 133.5855,B 0.9394,C -0.0445,E1 0.832,E2 321.3303} C_DIS
LIN {X -99.7719,Y 99.8885,Z 191,A 131.5881,B 0.9393,C -0.0476,E1 0.836,E2 323.3462} C_DIS
LIN {X -96.6064,Y 102.9532,Z 191,A 129.6186,B 0.9391,C -0.0506,E1 0.84,E2 325.3352} C_DIS
LIN {X -93.2416,Y 106.01,Z 191,A 127.6444,B 0.939,C -0.0535,E1 0.8442,E2 327.3229} C_DIS
LIN {X -90.1463,Y 108.6539,Z 191,A 125.8032,B 0.9388,C -0.0559,E1 0.8482,E2 329.1845} C_DIS
LIN {X -86.4472,Y 111.6194,Z 191,A 123.7468,B 0.9387,C -0.0586,E1 0.8528,E2 331.2546} C_DIS
LIN {X -82.7684,Y 114.374,Z 191,A 121.4175,B 0.9385,C -0.0608,E1 0.8582,E2 333.6345} C_DIS
LIN {X -79.6691,Y 116.5543,Z 191,A 120.0472,B 0.9384,C -0.0628,E1 0.8614,E2 334.9853} C_DIS
LIN {X -75.8011,Y 119.1064,Z 191,A 118.0461,B 0.9383,C -0.0649,E1 0.8662,E2 336.9987} C_DIS
LIN {X -71.9119,Y 121.4943,Z 191,A 115.5611,B 0.9381,C -0.0664,E1 0.8724,E2 339.5524} C_DIS
LIN {X -67.6236,Y 123.9317,Z 191,A 114.2478,B 0.938,C -0.0689,E1 0.8754,E2 340.7887} C_DIS
LIN {X -64.8293,Y 125.4167,Z 191,A 112.4348,B 0.938,C -0.0696,E1 0.8801,E2 342.6595} C_DIS
LIN {X -60.1115,Y 127.7448,Z 191,A 110.4863,B 0.9378,C -0.0715,E1 0.885,E2 344.5863} C_DIS
LIN {X -57.204,Y 129.0712,Z 191,A 108.7539,B 0.9378,C -0.072,E1 0.8896,E2 346.3657} C_DIS
LIN {X -53.6616,Y 130.5853,Z 191,A 107.5268,B 0.9376,C -0.0734,E1 0.8927,E2 347.5552} C_DIS
LIN {X -50.5886,Y 131.8052,Z 191,A 106.1616,B 0.9376,C -0.0741,E1 0.8963,E2 348.9223} C_DIS
LIN {X -47.774,Y 132.85,Z 191,A 104.8434,B 0.9376,C -0.0746,E1 0.8999,E2 350.2508} C_DIS
LIN {X -44.3423,Y 134.0347,Z 191,A 103.3668,B 0.9375,C -0.0753,E1 0.9038,E2 351.7269} C_DIS
LIN {X -41.1848,Y 135.0382,Z 191,A 101.9982,B 0.9375,C -0.0758,E1 0.9075,E2 353.0975} C_DIS
LIN {X -37.9577,Y 135.9805,Z 191,A 100.6055,B 0.9375,C -0.0761,E1 0.9113,E2 354.4926} C_DIS
LIN {X -33.917,Y 137.0469,Z 191,A 98.8917,B 0.9374,C -0.0765,E1 0.916,E2 356.2078} C_DIS
LIN {X -30.8046,Y 137.7788,Z 191,A 97.5958,B 0.9374,C -0.0767,E1 0.9196,E2 357.5028} C_DIS
LIN {X -28.1042,Y 138.3534,Z 191,A 96.4578,B 0.9374,C -0.0768,E1 0.9228,E2 358.6422} C_DIS
LIN {X -24.6811,Y 139.0051,Z 191,A 95.0283,B 0.9374,C -0.0768,E1 0.9268,E2 360.0727} C_DIS
LIN {X -21.004,Y 139.6092,Z 191,A 93.3773,B 0.9374,C -0.0765,E1 0.9314,E2 361.7382} C_DIS
LIN {X -14.9949,Y 140.3806,Z 191,A 91.0895,B 0.9374,C -0.0765,E1 0.9378,E2 364.0063} C_DIS
LIN {X -11.3279,Y 140.7251,Z 191,A 89.6159,B 0.9374,C -0.0762,E1 0.942,E2 365.477} C_DIS
LIN {X -7.2977,Y 140.9907,Z 191,A 87.9429,B 0.9374,C -0.0757,E1 0.9467,E2 367.153} C_DIS
LIN {X -3.435,Y 141.1384,Z 191,A 86.4074,B 0.9374,C -0.0751,E1 0.951,E2 368.6842} C_DIS
LIN {X 0.6841,Y 141.1777,Z 191,A 84.7556,B 0.9375,C -0.0744,E1 0.9557,E2 370.3332} C_DIS
LIN {X 4.7946,Y 141.0996,Z 191,A 83.0457,B 0.9376,C -0.0734,E1 0.9606,E2 372.0471} C_DIS
LIN {X 9.1807,Y 140.8813,Z 191,A 81.4002,B 0.9376,C -0.0727,E1 0.9652,E2 373.677} C_DIS
LIN {X 13.3846,Y 140.5433,Z 191,A 79.799,B 0.9378,C -0.0717,E1 0.9696,E2 375.2654} C_DIS
LIN {X 17.1787,Y 140.1309,Z 191,A 78.412,B 0.9378,C -0.071,E1 0.9735,E2 376.6339} C_DIS
LIN {X 19.9884,Y 139.757,Z 191,A 77.2391,B 0.9378,C -0.07,E1 0.9768,E2 377.8089} C_DIS
LIN {X 23.5297,Y 139.2048,Z 191,A 75.7803,B 0.938,C -0.0687,E1 0.9809,E2 379.2679} C_DIS
LIN {X 28.4774,Y 138.2775,Z 191,A 73.4754,B 0.9382,C -0.0659,E1 0.9873,E2 381.6011} C_DIS
LIN {X 32.6761,Y 137.3461,Z 191,A 72.4174,B 0.9382,C -0.0661,E1 0.9901,E2 382.5824} C_DIS
LIN {X 41.1637,Y 135.0446,Z 191,A 68.8276,B 0.9385,C -0.0619,E1 0.9998,E2 386.1737} C_DIS
LIN {X 44.3694,Y 134.0257,Z 191,A 67.5569,B 0.9385,C -0.0605,E1 1.0032,E2 387.4336} C_DIS
LIN {X 48.2739,Y 132.6698,Z 191,A 66.0752,B 0.9386,C -0.0589,E1 1.0071,E2 388.8929} C_DIS
LIN {X 51.4008,Y 131.4895,Z 191,A 64.7498,B 0.9388,C -0.0571,E1 1.0106,E2 390.2146} C_DIS
LIN {X 54.6824,Y 130.159,Z 191,A 63.4598,B 0.9388,C -0.0556,E1 1.0139,E2 391.4877} C_DIS
LIN {X 58.0246,Y 128.7042,Z 191,A 62.0906,B 0.939,C -0.0537,E1 1.0174,E2 392.8442} C_DIS
LIN {X 61.2506,Y 127.2006,Z 191,A 60.8196,B 0.939,C -0.0521,E1 1.0206,E2 394.0952} C_DIS
LIN {X 64.8293,Y 125.4167,Z 191,A 59.2737,B 0.9392,C -0.0498,E1 1.0245,E2 395.6323} C_DIS
LIN {X 69.2441,Y 123.0336,Z 191,A 57.344,B 0.9393,C -0.0468,E1 1.0292,E2 397.5496} C_DIS
LIN {X 73.2509,Y 120.6912,Z 191,A 55.6773,B 0.9394,C -0.0443,E1 1.0332,E2 399.1912} C_DIS
LIN {X 76.7076,Y 118.5242,Z 191,A 54.0806,B 0.9396,C -0.0416,E1 1.037,E2 400.7809} C_DIS
LIN {X 80.2963,Y 116.1236,Z 191,A 52.3535,B 0.9397,C -0.0384,E1 1.041,E2 402.5051} C_DIS
LIN {X 83.7994,Y 113.6211,Z 191,A 50.9153,B 0.9397,C -0.0363,E1 1.0442,E2 403.9075} C_DIS
LIN {X 87.4987,Y 110.7976,Z 191,A 49.1734,B 0.9399,C -0.0331,E1 1.048,E2 405.6323} C_DIS
LIN {X 91.2419,Y 107.7357,Z 191,A 47.4971,B 0.94,C -0.0303,E1 1.0515,E2 407.275} C_DIS
LIN {X 94.4773,Y 104.9104,Z 191,A 45.9224,B 0.94,C -0.0274,E1 1.0548,E2 408.8299} C_DIS
LIN {X 99.0251,Y 100.6284,Z 191,A 43.8746,B 0.9402,C -0.0241,E1 1.0589,E2 410.8202} C_DIS
LIN {X 102.5903,Y 96.991,Z 191,A 41.7827,B 0.9402,C -0.0194,E1 1.063,E2 412.9152} C_DIS
LIN {X 105.5948,Y 93.7114,Z 191,A 40.1414,B 0.9404,C -0.0161,E1 1.066,E2 414.5372} C_DIS
LIN {X 108.6139,Y 90.1946,Z 191,A 38.5172,B 0.9404,C -0.0129,E1 1.0689,E2 416.1308} C_DIS
LIN {X 112.185,Y 85.7119,Z 191,A 36.5689,B 0.9404,C -0.0091,E1 1.0722,E2 418.0338} C_DIS
LIN {X 114.419,Y 82.7063,Z 191,A 35.0325,B 0.9404,C -0.0054,E1 1.0748,E2 419.5725} C_DIS
LIN {X 116.9041,Y 79.1546,Z 191,A 33.2784,B 0.9404,C -0.0012,E1 1.0775,E2 421.3263} C_DIS
LIN {X 118.9436,Y 76.0555,Z 191,A 32.3305,B 0.9404,C -0.0001,E1 1.0789,E2 422.2064} C_DIS
LIN {X 120.8353,Y 73.0127,Z 191,A 30.9028,B 0.9404,C 0.0034,E1 1.081,E2 423.6312} C_DIS
LIN {X 123.0252,Y 69.2592,Z 191,A 29.3345,B 0.9404,C 0.0069,E1 1.0831,E2 425.1759} C_DIS
LIN {X 125.1872,Y 65.2669,Z 191,A 27.7795,B 0.9404,C 0.0102,E1 1.0851,E2 426.6957} C_DIS
LIN {X 126.9545,Y 61.7623,Z 191,A 26.2877,B 0.9404,C 0.0138,E1 1.0869,E2 428.1756} C_DIS
LIN {X 129.3543,Y 56.5619,Z 191,A 24.449,B 0.9404,C 0.0175,E1 1.089,E2 429.9541} C_DIS
LIN {X 131.1454,Y 52.2745,Z 191,A 22.7096,B 0.9402,C 0.0218,E1 1.0908,E2 431.6757} C_DIS
LIN {X 132.3451,Y 49.1567,Z 191,A 21.534,B 0.9402,C 0.0245,E1 1.092,E2 432.8291} C_DIS
LIN {X 133.4708,Y 46.0116,Z 191,A 20.3115,B 0.9401,C 0.0274,E1 1.0931,E2 434.0351} C_DIS
LIN {X 134.5861,Y 42.64,Z 191,A 19.0263,B 0.94,C 0.0305,E1 1.0942,E2 435.301} C_DIS
LIN {X 136.8167,Y 34.8238,Z 191,A 16.4291,B 0.9398,C 0.0359,E1 1.0961,E2 437.8098} C_DIS
LIN {X 138.2258,Y 28.7316,Z 191,A 14.0613,B 0.9396,C 0.042,E1 1.0976,E2 440.1569} C_DIS
LIN {X 139.3337,Y 22.7573,Z 191,A 11.8773,B 0.9393,C 0.0473,E1 1.0986,E2 442.3055} C_DIS
LIN {X 139.796,Y 19.7152,Z 191,A 10.7632,B 0.9392,C 0.0501,E1 1.0991,E2 443.4025} C_DIS
LIN {X 140.2817,Y 15.9141,Z 191,A 9.2678,B 0.9389,C 0.0541,E1 1.0996,E2 444.891} C_DIS
LIN {X 140.699,Y 11.6372,Z 191,A 7.8143,B 0.9387,C 0.0574,E1 1.0999,E2 446.3073} C_DIS
LIN {X 140.982,Y 7.4708,Z 191,A 6.342,B 0.9385,C 0.061,E1 1.1002,E2 447.7512} C_DIS
LIN {X 141.1365,Y 3.5013,Z 191,A 4.9231,B 0.9383,C 0.0644,E1 1.1002,E2 449.1454} C_DIS
LIN {X 141.1793,Y -0.6144,Z 191,A 3.4485,B 0.938,C 0.0681,E1 1.1002,E2 450.5949} C_DIS
LIN {X 141.1086,Y -4.5041,Z 191,A 2.0463,B 0.9378,C 0.0715,E1 1.1002,E2 451.9745} C_DIS
LIN {X 140.918,Y -8.5861,Z 191,A 0.7001,B 0.9375,C 0.0745,E1 1.1,E2 453.2799} C_DIS
LIN {X 140.6344,Y -12.4025,Z 191,A -0.6023,B 0.9373,C 0.0775,E1 1.0997,E2 454.5496} C_DIS
LIN {X 140.3271,Y -15.4926,Z 191,A -1.8428,B 0.937,C 0.0809,E1 1.0994,E2 455.7882} C_DIS
LIN {X 139.788,Y -19.771,Z 191,A -3.3836,B 0.9367,C 0.0846,E1 1.0988,E2 457.3018} C_DIS
LIN {X 139.0707,Y -24.3142,Z 191,A -4.9827,B 0.9363,C 0.0884,E1 1.0981,E2 458.8658} C_DIS
LIN {X 138.3259,Y -28.2398,Z 191,A -6.3693,B 0.936,C 0.0916,E1 1.0973,E2 460.2214} C_DIS
LIN {X 137.291,Y -32.9046,Z 191,A -7.9117,B 0.9357,C 0.0948,E1 1.0964,E2 461.7108} C_DIS
LIN {X 136.1342,Y -37.4083,Z 191,A -9.592,B 0.9353,C 0.0988,E1 1.0953,E2 463.364} C_DIS
LIN {X 135.28,Y -40.3901,Z 191,A -11.0258,B 0.9348,C 0.1032,E1 1.0941,E2 464.8227} C_DIS
LIN {X 134.2618,Y -43.6547,Z 191,A -12.0386,B 0.9346,C 0.1049,E1 1.0933,E2 465.7848} C_DIS
LIN {X 133.2431,Y -46.6686,Z 191,A -13.1024,B 0.9344,C 0.1072,E1 1.0923,E2 466.8179} C_DIS
LIN {X 131.9335,Y -50.2557,Z 191,A -14.4643,B 0.934,C 0.1103,E1 1.091,E2 468.1549} C_DIS
LIN {X 130.7645,Y -53.2196,Z 191,A -15.6254,B 0.9337,C 0.113,E1 1.0898,E2 469.2985} C_DIS
LIN {X 129.0983,Y -57.1435,Z 191,A -17.0779,B 0.9333,C 0.1161,E1 1.0883,E2 470.7135} C_DIS
LIN {X 126.26,Y -63.1701,Z 191,A -19.5019,B 0.9326,C 0.1216,E1 1.0854,E2 473.1003} C_DIS
LIN {X 124.3787,Y -66.7978,Z 191,A -21.1745,B 0.932,C 0.1259,E1 1.0832,E2 474.7761} C_DIS
LIN {X 122.4707,Y -70.2356,Z 191,A -22.996,B 0.9313,C 0.1311,E1 1.0806,E2 476.6306} C_DIS
LIN {X 119.4882,Y -75.1972,Z 191,A -24.5356,B 0.9311,C 0.1328,E1 1.0785,E2 478.0578} C_DIS
LIN {X 117.0006,Y -79.012,Z 191,A -26.1755,B 0.9306,C 0.1363,E1 1.076,E2 479.6695} C_DIS
LIN {X 114.4537,Y -82.6584,Z 191,A -27.78,B 0.9301,C 0.1396,E1 1.0734,E2 481.2467} C_DIS
LIN {X 111.7754,Y -86.2459,Z 191,A -29.4017,B 0.9296,C 0.1429,E1 1.0707,E2 482.8419} C_DIS
LIN {X 108.8429,Y -89.918,Z 191,A -31.0818,B 0.9291,C 0.1462,E1 1.0678,E2 484.4909} C_DIS
LIN {X 106.0252,Y -93.2244,Z 191,A -32.66,B 0.9286,C 0.1493,E1 1.065,E2 486.0439} C_DIS
LIN {X 102.9721,Y -96.5863,Z 191,A -34.3204,B 0.928,C 0.1525,E1 1.0619,E2 487.6794} C_DIS
LIN {X 99.7519,Y -99.9083,Z 191,A -36.0125,B 0.9275,C 0.1557,E1 1.0586,E2 489.346} C_DIS
LIN {X 96.4894,Y -103.0628,Z 191,A -37.6254,B 0.927,C 0.1586,E1 1.0554,E2 490.9272} C_DIS
LIN {X 93.2416,Y -106.01,Z 191,A -39.2468,B 0.9265,C 0.1615,E1 1.052,E2 492.527} C_DIS
LIN {X 89.7423,Y -108.9884,Z 191,A -40.938,B 0.926,C 0.1645,E1 1.0484,E2 494.1943} C_DIS
LIN {X 86.1232,Y -111.8704,Z 191,A -42.6595,B 0.9255,C 0.1675,E1 1.0446,E2 495.8944} C_DIS
LIN {X 82.3888,Y -114.6482,Z 191,A -44.3646,B 0.925,C 0.1702,E1 1.0408,E2 497.574} C_DIS
LIN {X 78.578,Y -117.2926,Z 191,A -46.026,B 0.9245,C 0.1727,E1 1.037,E2 499.2044} C_DIS
LIN {X 74.9124,Y -119.6674,Z 191,A -47.6284,B 0.924,C 0.1752,E1 1.0333,E2 500.7831} C_DIS
LIN {X 71.2408,Y -121.8887,Z 191,A -49.2833,B 0.9235,C 0.1778,E1 1.0293,E2 502.4266} C_DIS
LIN {X 64.6161,Y -125.5253,Z 191,A -51.9209,B 0.9229,C 0.181,E1 1.0229,E2 505.003} C_DIS
LIN {X 61.9422,Y -126.8658,Z 191,A -53.6636,B 0.9221,C 0.1851,E1 1.0183,E2 506.8248} C_DIS
LIN {X 57.328,Y -129.0157,Z 191,A -55.0455,B 0.9221,C 0.1854,E1 1.015,E2 508.107} C_DIS
LIN {X 54.1427,Y -130.3844,Z 191,A -56.3635,B 0.9217,C 0.1871,E1 1.0116,E2 509.4128} C_DIS
LIN {X 51.0318,Y -131.6329,Z 191,A -57.6271,B 0.9214,C 0.1886,E1 1.0083,E2 510.6629} C_DIS
LIN {X 47.3926,Y -132.9875,Z 191,A -59.0616,B 0.9211,C 0.1902,E1 1.0046,E2 512.0775} C_DIS
LIN {X 44.0219,Y -134.1414,Z 191,A -60.8219,B 0.9204,C 0.1932,E1 0.9997,E2 513.8857} C_DIS
LIN {X 40.0807,Y -135.3706,Z 191,A -61.9619,B 0.9204,C 0.1932,E1 0.9969,E2 514.947} C_DIS
LIN {X 37.555,Y -136.0932,Z 191,A -63.1486,B 0.9201,C 0.1949,E1 0.9936,E2 516.1524} C_DIS
LIN {X 31.6889,Y -137.5769,Z 191,A -65.1162,B 0.9199,C 0.1958,E1 0.9884,E2 518.0485} C_DIS
LIN {X 25.2683,Y -138.9,Z 191,A -67.6911,B 0.9194,C 0.1981,E1 0.9813,E2 520.6124} C_DIS
LIN {X 20.8044,Y -139.6401,Z 191,A -69.7585,B 0.9189,C 0.2005,E1 0.9754,E2 522.7158} C_DIS
LIN {X 16.448,Y -140.218,Z 191,A -71.2994,B 0.9187,C 0.2011,E1 0.9712,E2 524.2213} C_DIS
LIN {X 12.464,Y -140.6292,Z 191,A -72.9443,B 0.9185,C 0.2024,E1 0.9665,E2 525.8701} C_DIS
LIN {X 8.5242,Y -140.9218,Z 191,A -74.4381,B 0.9183,C 0.2031,E1 0.9623,E2 527.3483} C_DIS
LIN {X 5.3337,Y -141.0786,Z 191,A -75.6289,B 0.9183,C 0.2035,E1 0.959,E2 528.524} C_DIS
LIN {X 2.3206,Y -141.1603,Z 191,A -76.8698,B 0.9181,C 0.2042,E1 0.9555,E2 529.7682} C_DIS
LIN {X 2.3206,Y -141.1603,Z 191,A -76.8698,B 0.9181,C 0.2042,E1 0.9555,E2 529.7682} C_DIS
Enddeposition()
LIN {X 1.0182,Y -142.072,Z 191,A -76.8746,B 0.9184,C 0.2033,E1 0.9558,E2 529.7177} C_DIS
Startdeposition()
$VEL.CP = VEL_PRINT
LIN {X 4.2568,Y -142.0148,Z 191,A -75.5387,B 0.9186,C 0.2025,E1 0.9595,E2 528.3766} C_DIS
LIN {X 7.2811,Y -141.8916,Z 191,A -74.3451,B 0.9186,C 0.2019,E1 0.9629,E2 527.1865} C_DIS
LIN {X 11.1149,Y -141.6448,Z 191,A -72.7203,B 0.919,C 0.2006,E1 0.9675,E2 525.5492} C_DIS
LIN {X 15.1711,Y -141.2658,Z 191,A -71.2163,B 0.9191,C 0.1999,E1 0.9717,E2 524.0654} C_DIS
LIN {X 18.5677,Y -140.8596,Z 191,A -69.9512,B 0.9193,C 0.1991,E1 0.9752,E2 522.8169} C_DIS
LIN {X 21.5443,Y -140.4352,Z 191,A -68.8502,B 0.9194,C 0.1985,E1 0.9783,E2 521.7321} C_DIS
LIN {X 24.3001,Y -139.9864,Z 191,A -67.7321,B 0.9196,C 0.1975,E1 0.9814,E2 520.6145} C_DIS
LIN {X 28.4288,Y -139.2047,Z 191,A -65.7368,B 0.9202,C 0.1948,E1 0.987,E2 518.5723} C_DIS
LIN {X 32.2471,Y -138.3714,Z 191,A -64.5409,B 0.9202,C 0.1945,E1 0.9902,E2 517.4334} C_DIS
LIN {X 36.0084,Y -137.4405,Z 191,A -63.179,B 0.9205,C 0.1935,E1 0.9938,E2 516.101} C_DIS
LIN {X 39.4977,Y -136.478,Z 191,A -61.7971,B 0.9208,C 0.1921,E1 0.9976,E2 514.7298} C_DIS
LIN {X 44.6051,Y -134.8947,Z 191,A -59.661,B 0.9213,C 0.1895,E1 1.0033,E2 512.5953} C_DIS
LIN {X 48.2766,Y -133.6244,Z 191,A -58.2807,B 0.9216,C 0.1882,E1 1.0069,E2 511.2421} C_DIS
LIN {X 51.1482,Y -132.5521,Z 191,A -57.0708,B 0.9219,C 0.1866,E1 1.0101,E2 510.0353} C_DIS
LIN {X 54.85,Y -131.0632,Z 191,A -55.2527,B 0.9225,C 0.1835,E1 1.0149,E2 508.1844} C_DIS
LIN {X 58.5047,Y -129.4741,Z 191,A -53.9912,B 0.9227,C 0.1825,E1 1.018,E2 506.974} C_DIS
LIN {X 62.7434,Y -127.4729,Z 191,A -52.4172,B 0.9231,C 0.1809,E1 1.0219,E2 505.4463} C_DIS
LIN {X 65.9369,Y -125.8507,Z 191,A -50.8477,B 0.9236,C 0.178,E1 1.0259,E2 503.857} C_DIS
LIN {X 70.4239,Y -123.3982,Z 191,A -49.08,B 0.924,C 0.1758,E1 1.0301,E2 502.1321} C_DIS
LIN {X 74.2669,Y -121.1242,Z 191,A -47.4234,B 0.9245,C 0.1733,E1 1.0341,E2 500.4957} C_DIS
LIN {X 78.0634,Y -118.7128,Z 191,A -45.7755,B 0.925,C 0.1708,E1 1.0379,E2 498.8713} C_DIS
LIN {X 81.7259,Y -116.222,Z 191,A -44.1241,B 0.9255,C 0.1681,E1 1.0417,E2 497.2386} C_DIS
LIN {X 85.1169,Y -113.7623,Z 191,A -42.5739,B 0.9259,C 0.1655,E1 1.0452,E2 495.708} C_DIS
LIN {X 88.871,Y -110.8546,Z 191,A -40.8478,B 0.9265,C 0.1626,E1 1.0489,E2 494.0085} C_DIS
LIN {X 92.4272,Y -107.9074,Z 191,A -39.1622,B 0.927,C 0.1596,E1 1.0525,E2 492.3478} C_DIS
LIN {X 95.8844,Y -104.8472,Z 191,A -37.4786,B 0.9275,C 0.1566,E1 1.056,E2 490.6891} C_DIS
LIN {X 99.3247,Y -101.5938,Z 191,A -35.7742,B 0.928,C 0.1535,E1 1.0594,E2 489.0136} C_DIS
LIN {X 102.7186,Y -98.1607,Z 191,A -34.0532,B 0.9285,C 0.1503,E1 1.0627,E2 487.3243} C_DIS
LIN {X 105.9107,Y -94.7078,Z 191,A -32.3522,B 0.929,C 0.147,E1 1.0658,E2 485.6505} C_DIS
LIN {X 108.9857,Y -91.1526,Z 191,A -30.6579,B 0.9296,C 0.1437,E1 1.0689,E2 483.9843} C_DIS
LIN {X 111.8992,Y -87.5516,Z 191,A -28.9929,B 0.9301,C 0.1404,E1 1.0717,E2 482.3475} C_DIS
LIN {X 114.5919,Y -83.9962,Z 191,A -27.4066,B 0.9306,C 0.1372,E1 1.0743,E2 480.7907} C_DIS
LIN {X 117.1723,Y -80.3572,Z 191,A -25.8306,B 0.931,C 0.134,E1 1.0768,E2 479.2458} C_DIS
LIN {X 119.5773,Y -76.7328,Z 191,A -24.3895,B 0.9314,C 0.1313,E1 1.0789,E2 477.8487} C_DIS
LIN {X 121.84,Y -73.087,Z 191,A -22.4653,B 0.9321,C 0.126,E1 1.0818,E2 475.8952} C_DIS
LIN {X 123.817,Y -69.685,Z 191,A -21.3471,B 0.9323,C 0.1244,E1 1.0832,E2 474.8434} C_DIS
LIN {X 125.8389,Y -65.9592,Z 191,A -19.8885,B 0.9327,C 0.1214,E1 1.0851,E2 473.4195} C_DIS
LIN {X 127.431,Y -62.8284,Z 191,A -18.3423,B 0.9333,C 0.117,E1 1.0871,E2 471.8536} C_DIS
LIN {X 129.0484,Y -59.4359,Z 191,A -17.3652,B 0.9334,C 0.1159,E1 1.0881,E2 470.9525} C_DIS
LIN {X 130.4849,Y -56.2121,Z 191,A -15.9796,B 0.9339,C 0.1124,E1 1.0897,E2 469.5712} C_DIS
LIN {X 132.0357,Y -52.4704,Z 191,A -14.6311,B 0.9342,C 0.1096,E1 1.091,E2 468.262} C_DIS
LIN {X 133.4705,Y -48.7032,Z 191,A -13.1349,B 0.9346,C 0.106,E1 1.0925,E2 466.783} C_DIS
LIN {X 134.6627,Y -45.3017,Z 191,A -11.3277,B 0.9353,C 0.1002,E1 1.0941,E2 464.9246} C_DIS
LIN {X 136.3646,Y -39.8851,Z 191,A -9.931,B 0.9354,C 0.0988,E1 1.0952,E2 463.6525} C_DIS
LIN {X 137.93,Y -34.0897,Z 191,A -7.824,B 0.9359,C 0.0939,E1 1.0966,E2 461.5879} C_DIS
LIN {X 138.6119,Y -31.1945,Z 191,A -6.7833,B 0.9362,C 0.0914,E1 1.0973,E2 460.5684} C_DIS
LIN {X 139.1987,Y -28.4586,Z 191,A -5.8495,B 0.9364,C 0.0894,E1 1.0978,E2 459.6609} C_DIS
LIN {X 139.75,Y -25.6212,Z 191,A -4.8386,B 0.9366,C 0.087,E1 1.0983,E2 458.6708} C_DIS
LIN {X 140.1944,Y -23.0607,Z 191,A -3.8867,B 0.9368,C 0.0846,E1 1.0987,E2 457.7315} C_DIS
LIN {X 140.771,Y -19.2438,Z 191,A -2.5089,B 0.9371,C 0.0813,E1 1.0993,E2 456.3774} C_DIS
LIN {X 141.1372,Y -16.3314,Z 191,A -1.473,B 0.9373,C 0.0788,E1 1.0996,E2 455.361} C_DIS
LIN {X 141.5334,Y -12.4393,Z 191,A 0.0046,B 0.9376,C 0.0749,E1 1.1,E2 453.8962} C_DIS
LIN {X 141.8065,Y -8.7826,Z 191,A 1.1627,B 0.9378,C 0.0725,E1 1.1002,E2 452.781} C_DIS
LIN {X 141.9615,Y -5.7614,Z 191,A 2.2912,B 0.938,C 0.0696,E1 1.1003,E2 451.6643} C_DIS
LIN {X 142.0671,Y -1.8527,Z 191,A 3.6149,B 0.9383,C 0.0666,E1 1.1004,E2 450.3741} C_DIS
LIN {X 142.0605,Y 2.2465,Z 191,A 5.0523,B 0.9385,C 0.0631,E1 1.1004,E2 448.965} C_DIS
LIN {X 141.982,Y 5.2354,Z 191,A 6.1031,B 0.9387,C 0.0606,E1 1.1004,E2 447.9343} C_DIS
LIN {X 141.8395,Y 8.2468,Z 191,A 7.2051,B 0.9388,C 0.0578,E1 1.1001,E2 446.847} C_DIS
LIN {X 141.5979,Y 11.6758,Z 191,A 8.4377,B 0.939,C 0.0547,E1 1.0999,E2 445.6343} C_DIS
LIN {X 141.2878,Y 14.9666,Z 191,A 9.5168,B 0.9392,C 0.0524,E1 1.0996,E2 444.5884} C_DIS
LIN {X 140.9523,Y 17.8604,Z 191,A 10.5482,B 0.9392,C 0.0499,E1 1.0992,E2 443.5755} C_DIS
LIN {X 140.5485,Y 20.8036,Z 191,A 11.7556,B 0.9395,C 0.0465,E1 1.0988,E2 442.3664} C_DIS
LIN {X 139.6864,Y 25.9688,Z 191,A 13.6684,B 0.9397,C 0.0417,E1 1.0978,E2 440.479} C_DIS
LIN {X 138.6672,Y 30.9524,Z 191,A 15.3316,B 0.9398,C 0.0381,E1 1.0969,E2 438.8662} C_DIS
LIN {X 137.7887,Y 34.6482,Z 191,A 16.6322,B 0.94,C 0.0351,E1 1.0961,E2 437.5951} C_DIS
LIN {X 136.5663,Y 39.1961,Z 191,A 18.5107,B 0.9401,C 0.0301,E1 1.0946,E2 435.7187} C_DIS
LIN {X 135.6064,Y 42.3998,Z 191,A 19.5732,B 0.9401,C 0.0279,E1 1.0938,E2 434.693} C_DIS
LIN {X 134.3119,Y 46.3297,Z 191,A 20.9161,B 0.9403,C 0.0251,E1 1.0926,E2 433.3916} C_DIS
LIN {X 132.5355,Y 51.191,Z 191,A 22.8028,B 0.9403,C 0.0205,E1 1.0908,E2 431.5301} C_DIS
LIN {X 131.2061,Y 54.5079,Z 191,A 23.9464,B 0.9404,C 0.0182,E1 1.0896,E2 430.4242} C_DIS
LIN {X 130.0584,Y 57.1984,Z 191,A 25.1508,B 0.9404,C 0.015,E1 1.0883,E2 429.2163} C_DIS
LIN {X 128.3494,Y 60.9312,Z 191,A 26.5115,B 0.9405,C 0.0122,E1 1.0867,E2 427.8927} C_DIS
LIN {X 126.9681,Y 63.7633,Z 191,A 27.6533,B 0.9405,C 0.0095,E1 1.0853,E2 426.7669} C_DIS
LIN {X 124.9911,Y 67.5573,Z 191,A 29.1819,B 0.9405,C 0.0061,E1 1.0833,E2 425.2628} C_DIS
LIN {X 122.8531,Y 71.3708,Z 191,A 30.7684,B 0.9406,C 0.0025,E1 1.0812,E2 423.6982} C_DIS
LIN {X 120.4548,Y 75.3484,Z 191,A 32.3138,B 0.9406,C -0.0006,E1 1.079,E2 422.1935} C_DIS
LIN {X 118.3836,Y 78.5627,Z 191,A 33.7858,B 0.9406,C -0.0041,E1 1.0767,E2 420.73} C_DIS
LIN {X 115.8755,Y 82.2171,Z 191,A 35.3384,B 0.9406,C -0.0073,E1 1.0743,E2 419.2062} C_DIS
LIN {X 113.2437,Y 85.8055,Z 191,A 36.9644,B 0.9406,C -0.0108,E1 1.0716,E2 417.6009} C_DIS
LIN {X 110.5619,Y 89.234,Z 191,A 38.4722,B 0.9406,C -0.0138,E1 1.069,E2 416.1234} C_DIS
LIN {X 107.9489,Y 92.3789,Z 191,A 39.9505,B 0.9405,C -0.0168,E1 1.0664,E2 414.6659} C_DIS
LIN {X 104.9934,Y 95.7242,Z 191,A 41.522,B 0.9405,C -0.0198,E1 1.0635,E2 413.1222} C_DIS
LIN {X 102.0668,Y 98.8383,Z 191,A 43.1191,B 0.9403,C -0.0231,E1 1.0604,E2 411.5403} C_DIS
LIN {X 99.7519,Y 101.1747,Z 191,A 44.3931,B 0.9403,C -0.0257,E1 1.0579,E2 410.2726} C_DIS
LIN {X 96.2036,Y 104.5538,Z 191,A 46.0527,B 0.9402,C -0.0286,E1 1.0546,E2 408.6512} C_DIS
LIN {X 93.194,Y 107.2455,Z 191,A 47.5141,B 0.9401,C -0.0313,E1 1.0515,E2 407.2098} C_DIS
LIN {X 90.1039,Y 109.8544,Z 191,A 49.0188,B 0.94,C -0.034,E1 1.0483,E2 405.7203} C_DIS
LIN {X 86.6086,Y 112.6309,Z 191,A 50.6096,B 0.9399,C -0.0367,E1 1.0448,E2 404.1545} C_DIS
LIN {X 83.6542,Y 114.8422,Z 191,A 51.9652,B 0.9398,C -0.0391,E1 1.0418,E2 402.8147} C_DIS
LIN {X 80.1315,Y 117.3272,Z 191,A 53.4892,B 0.9397,C -0.0415,E1 1.0383,E2 401.3163} C_DIS
LIN {X 77.0822,Y 119.3528,Z 191,A 54.942,B 0.9396,C -0.0441,E1 1.0349,E2 399.8664} C_DIS
LIN {X 73.201,Y 121.7719,Z 191,A 56.6229,B 0.9394,C -0.0467,E1 1.0309,E2 398.2049} C_DIS
LIN {X 69.1885,Y 124.0958,Z 191,A 58.3491,B 0.9394,C -0.0494,E1 1.0267,E2 396.4958} C_DIS
LIN {X 64.7797,Y 126.4507,Z 191,A 59.9769,B 0.9392,C -0.0512,E1 1.0228,E2 394.9136} C_DIS
LIN {X 61.8029,Y 127.9329,Z 191,A 61.3899,B 0.9391,C -0.0536,E1 1.0192,E2 393.4924} C_DIS
LIN {X 58.4264,Y 129.5092,Z 191,A 62.6479,B 0.9391,C -0.055,E1 1.016,E2 392.263} C_DIS
LIN {X 55.6042,Y 130.7477,Z 191,A 64.01,B 0.9389,C -0.0573,E1 1.0125,E2 390.8873} C_DIS
LIN {X 51.2762,Y 132.5024,Z 191,A 65.6648,B 0.9388,C -0.0591,E1 1.0082,E2 389.2592} C_DIS
LIN {X 47.128,Y 134.0352,Z 191,A 67.3439,B 0.9386,C -0.0611,E1 1.0038,E2 387.5927} C_DIS
LIN {X 44.1364,Y 135.0507,Z 191,A 68.8621,B 0.9385,C -0.0636,E1 0.9996,E2 386.0466} C_DIS
LIN {X 40.2938,Y 136.2449,Z 191,A 69.8178,B 0.9385,C -0.0634,E1 0.9972,E2 385.1679} C_DIS
LIN {X 36.9713,Y 137.1837,Z 191,A 71.1228,B 0.9384,C -0.0647,E1 0.9937,E2 383.8733} C_DIS
LIN {X 33.9021,Y 137.9753,Z 191,A 72.5401,B 0.9383,C -0.0666,E1 0.9898,E2 382.4404} C_DIS
LIN {X 29.8471,Y 138.9075,Z 191,A 74.185,B 0.9381,C -0.0682,E1 0.9852,E2 380.7997} C_DIS
LIN {X 25.3305,Y 139.802,Z 191,A 75.9258,B 0.9381,C -0.0696,E1 0.9804,E2 379.0726} C_DIS
LIN {X 21.5454,Y 140.435,Z 191,A 77.3584,B 0.938,C -0.0707,E1 0.9765,E2 377.6535} C_DIS
LIN {X 17.4458,Y 141.0043,Z 191,A 78.9104,B 0.9379,C -0.0717,E1 0.9722,E2 376.1154} C_DIS
LIN {X 13.7963,Y 141.4069,Z 191,A 80.2936,B 0.9379,C -0.0726,E1 0.9683,E2 374.7437} C_DIS
LIN {X 10.8447,Y 141.6646,Z 191,A 81.4449,B 0.9378,C -0.0733,E1 0.9651,E2 373.5977} C_DIS
LIN {X 7.7556,Y 141.8677,Z 191,A 82.6196,B 0.9378,C -0.0739,E1 0.9618,E2 372.4317} C_DIS
LIN {X 4.8459,Y 141.9972,Z 191,A 83.8155,B 0.9376,C -0.0746,E1 0.9584,E2 371.2338} C_DIS
LIN {X 1.1298,Y 142.0742,Z 191,A 85.3381,B 0.9376,C -0.0754,E1 0.9541,E2 369.7091} C_DIS
LIN {X -2.8882,Y 142.0499,Z 191,A 86.8835,B 0.9376,C -0.0759,E1 0.9497,E2 368.1728} C_DIS
LIN {X -6.6458,Y 141.9235,Z 191,A 88.2366,B 0.9376,C -0.0761,E1 0.9459,E2 366.8385} C_DIS
LIN {X -9.2861,Y 141.7755,Z 191,A 89.3912,B 0.9375,C -0.0766,E1 0.9426,E2 365.6745} C_DIS
LIN {X -12.3033,Y 141.5449,Z 191,A 90.6331,B 0.9375,C -0.077,E1 0.9391,E2 364.4307} C_DIS
LIN {X -15.3186,Y 141.2499,Z 191,A 91.8431,B 0.9375,C -0.0772,E1 0.9357,E2 363.2225} C_DIS
LIN {X -19.5795,Y 140.7235,Z 191,A 93.5124,B 0.9375,C -0.0772,E1 0.9311,E2 361.5609} C_DIS
LIN {X -22.4637,Y 140.2929,Z 191,A 94.9043,B 0.9374,C -0.0777,E1 0.9271,E2 360.1453} C_DIS
LIN {X -26.3737,Y 139.609,Z 191,A 96.2398,B 0.9374,C -0.0771,E1 0.9235,E2 358.8402} C_DIS
LIN {X -28.8569,Y 139.1176,Z 191,A 97.4072,B 0.9374,C -0.0773,E1 0.9202,E2 357.6569} C_DIS
LIN {X -32.847,Y 138.2296,Z 191,A 99.0374,B 0.9374,C -0.077,E1 0.9157,E2 356.0295} C_DIS
LIN {X -35.9322,Y 137.4609,Z 191,A 100.4449,B 0.9374,C -0.0769,E1 0.9118,E2 354.6086} C_DIS
LIN {X -39.8506,Y 136.3747,Z 191,A 101.9331,B 0.9375,C -0.0762,E1 0.9078,E2 353.1381} C_DIS
LIN {X -42.9163,Y 135.4415,Z 191,A 103.2523,B 0.9375,C -0.0757,E1 0.9042,E2 351.8166} C_DIS
LIN {X -45.8879,Y 134.4651,Z 191,A 104.5356,B 0.9376,C -0.0752,E1 0.9007,E2 350.5316} C_DIS
LIN {X -49.3733,Y 133.2239,Z 191,A 106.2549,B 0.9376,C -0.0747,E1 0.8961,E2 348.7874} C_DIS
LIN {X -52.8497,Y 131.8828,Z 191,A 107.5979,B 0.9377,C -0.0736,E1 0.8926,E2 347.4631} C_DIS
LIN {X -55.9532,Y 130.5967,Z 191,A 108.9418,B 0.9377,C -0.0727,E1 0.8891,E2 346.1212} C_DIS
LIN {X -58.7609,Y 129.3596,Z 191,A 110.5717,B 0.9378,C -0.0723,E1 0.8848,E2 344.4477} C_DIS
LIN {X -63.7866,Y 126.9562,Z 191,A 112.8665,B 0.938,C -0.0705,E1 0.8789,E2 342.1486} C_DIS
LIN {X -67.2483,Y 125.1572,Z 191,A 114.598,B 0.938,C -0.0692,E1 0.8746,E2 340.4} C_DIS
LIN {X -71.5716,Y 122.7369,Z 191,A 116.5768,B 0.9382,C -0.0671,E1 0.8697,E2 338.4246} C_DIS
LIN {X -75.0282,Y 120.6541,Z 191,A 118.2895,B 0.9383,C -0.0654,E1 0.8656,E2 336.7031} C_DIS
LIN {X -78.3544,Y 118.5213,Z 191,A 119.968,B 0.9385,C -0.0636,E1 0.8616,E2 335.0158} C_DIS
LIN {X -81.5378,Y 116.3544,Z 191,A 121.761,B 0.9385,C -0.0618,E1 0.8573,E2 333.1962} C_DIS
LIN {X -85.3782,Y 113.5661,Z 191,A 123.8048,B 0.9387,C -0.0593,E1 0.8527,E2 331.1386} C_DIS
LIN {X -89.1076,Y 110.6638,Z 191,A 125.8153,B 0.9389,C -0.0567,E1 0.8482,E2 329.1171} C_DIS
LIN {X -92.4816,Y 107.8605,Z 191,A 127.8036,B 0.9391,C -0.0541,E1 0.8439,E2 327.1045} C_DIS
LIN {X -95.7574,Y 104.9633,Z 191,A 129.72,B 0.9392,C -0.0513,E1 0.8398,E2 325.1714} C_DIS
LIN {X -99.0476,Y 101.8641,Z 191,A 131.7076,B 0.9394,C -0.0483,E1 0.8357,E2 323.1657} C_DIS
LIN {X -102.2376,Y 98.6618,Z 191,A 133.7157,B 0.9395,C -0.0452,E1 0.8317,E2 321.1369} C_DIS
LIN {X -105.364,Y 95.3158,Z 191,A 135.7719,B 0.9397,C -0.0418,E1 0.8278,E2 319.0572} C_DIS
LIN {X -108.2976,Y 91.9688,Z 191,A 137.7519,B 0.9398,C -0.0384,E1 0.8241,E2 317.0565} C_DIS
LIN {X -111.0732,Y 88.5968,Z 191,A 139.7224,B 0.94,C -0.0349,E1 0.8205,E2 315.0623} C_DIS
LIN {X -112.8386,Y 86.3371,Z 191,A 141.0607,B 0.94,C -0.0325,E1 0.8182,E2 313.703} C_DIS
LIN {X -115.8763,Y 82.216,Z 191,A 143.3137,B 0.9402,C -0.0281,E1 0.8145,E2 311.4288} C_DIS
LIN {X -118.2453,Y 78.7699,Z 191,A 145.2797,B 0.9402,C -0.0244,E1 0.8113,E2 309.4301} C_DIS
LIN {X -120.6359,Y 75.0575,Z 191,A 147.298,B 0.9404,C -0.0203,E1 0.8082,E2 307.3843} C_DIS
LIN {X -123.2658,Y 70.656,Z 191,A 149.828,B 0.9404,C -0.0154,E1 0.8046,E2 304.7993} C_DIS
LIN {X -125.4551,Y 66.6902,Z 191,A 151.7763,B 0.9405,C -0.011,E1 0.802,E2 302.8371} C_DIS
LIN {X -127.2359,Y 63.2238,Z 191,A 154.0896,B 0.9405,C -0.0068,E1 0.799,E2 300.4331} C_DIS
LIN {X -129.2371,Y 59.0277,Z 191,A 155.7826,B 0.9406,C -0.0023,E1 0.797,E2 298.7639} C_DIS
LIN {X -131.1671,Y 54.6013,Z 191,A 158.0163,B 0.9406,C 0.0027,E1 0.7945,E2 296.4957} C_DIS
LIN {X -132.7021,Y 50.7624,Z 191,A 160.0468,B 0.9406,C 0.0072,E1 0.7924,E2 294.4209} C_DIS
LIN {X -134.0147,Y 47.1871,Z 191,A 161.5603,B 0.9406,C 0.0112,E1 0.791,E2 292.9111} C_DIS
LIN {X -135.2682,Y 43.4588,Z 191,A 163.2928,B 0.9405,C 0.0154,E1 0.7894,E2 291.1612} C_DIS
LIN {X -136.0887,Y 40.8239,Z 191,A 164.9448,B 0.9405,C 0.0188,E1 0.788,E2 289.4415} C_DIS
LIN {X -136.932,Y 37.8933,Z 191,A 167.0112,B 0.9403,C 0.0229,E1 0.7865,E2 287.2683} C_DIS
LIN {X -138.286,Y 32.6131,Z 191,A 168.7533,B 0.9402,C 0.0283,E1 0.7853,E2 285.5866} C_DIS
LIN {X -139.3819,Y 27.558,Z 191,A 171.4255,B 0.94,C 0.0346,E1 0.7838,E2 282.8399} C_DIS
LIN {X -140.5338,Y 20.9051,Z 191,A 174.586,B 0.9397,C 0.0425,E1 0.7823,E2 279.6241} C_DIS
LIN {X -141.0698,Y 16.8967,Z 191,A 176.2737,B 0.9394,C 0.047,E1 0.7817,E2 277.9298} C_DIS
LIN {X -141.3561,Y 14.3249,Z 191,A 177.5735,B 0.9393,C 0.0502,E1 0.7813,E2 276.597} C_DIS
LIN {X -141.679,Y 10.6466,Z 191,A 179.4614,B 0.939,C 0.0547,E1 0.7809,E2 274.6572} C_DIS
LIN {X -141.9533,Y 5.9727,Z 191,A -178.5458,B 0.9387,C 0.0601,E1 0.7806,E2 272.6515} C_DIS
LIN {X -142.0522,Y 2.7474,Z 191,A -176.7005,B 0.9384,C 0.0642,E1 0.7804,E2 270.7343} C_DIS
LIN {X -142.0576,Y -2.4245,Z 191,A -174.5033,B 0.938,C 0.0702,E1 0.7804,E2 268.5232} C_DIS
LIN {X -141.9943,Y -4.9206,Z 191,A -173.3063,B 0.9378,C 0.0731,E1 0.7806,E2 267.3013} C_DIS
LIN {X -141.8882,Y -7.3492,Z 191,A -172.0073,B 0.9375,C 0.0762,E1 0.7808,E2 265.9597} C_DIS
LIN {X -141.543,Y -12.3251,Z 191,A -169.5496,B 0.937,C 0.0822,E1 0.7813,E2 263.4422} C_DIS
LIN {X -141.0766,Y -16.8394,Z 191,A -167.4535,B 0.9365,C 0.0875,E1 0.782,E2 261.3106} C_DIS
LIN {X -140.5153,Y -21.027,Z 191,A -165.3361,B 0.9361,C 0.0925,E1 0.7828,E2 259.1372} C_DIS
LIN {X -139.8411,Y -25.112,Z 191,A -163.5473,B 0.9356,C 0.0972,E1 0.7837,E2 257.3326} C_DIS
LIN {X -138.9344,Y -29.7227,Z 191,A -161.5538,B 0.935,C 0.1024,E1 0.7848,E2 255.3263} C_DIS
LIN {X -138.1894,Y -33.0137,Z 191,A -159.8927,B 0.9346,C 0.1063,E1 0.7858,E2 253.624} C_DIS
LIN {X -137.2385,Y -36.7658,Z 191,A -157.9363,B 0.9341,C 0.1107,E1 0.7873,E2 251.6131} C_DIS
LIN {X -136.3919,Y -39.7918,Z 191,A -156.5063,B 0.9337,C 0.1141,E1 0.7884,E2 250.1608} C_DIS
LIN {X -135.5481,Y -42.5826,Z 191,A -154.9871,B 0.9333,C 0.1174,E1 0.7897,E2 248.5936} C_DIS
LIN {X -134.2934,Y -46.3832,Z 191,A -153.2598,B 0.9327,C 0.1217,E1 0.7912,E2 246.8508} C_DIS
LIN {X -133.3506,Y -49.0351,Z 191,A -151.8479,B 0.9323,C 0.1247,E1 0.7926,E2 245.4001} C_DIS
LIN {X -132.3676,Y -51.623,Z 191,A -150.6265,B 0.9319,C 0.1276,E1 0.7938,E2 244.1641} C_DIS
LIN {X -131.2944,Y -54.2964,Z 191,A -149.3566,B 0.9315,C 0.1305,E1 0.7952,E2 242.8792} C_DIS
LIN {X -129.0541,Y -59.4236,Z 191,A -146.4103,B 0.9307,C 0.1363,E1 0.7987,E2 239.8347} C_DIS
LIN {X -126.9797,Y -63.7405,Z 191,A -144.2284,B 0.93,C 0.141,E1 0.8014,E2 237.6172} C_DIS
LIN {X -125.0581,Y -67.4326,Z 191,A -142.3648,B 0.9294,C 0.145,E1 0.8039,E2 235.7273} C_DIS
LIN {X -122.9393,Y -71.222,Z 191,A -140.382,B 0.9287,C 0.149,E1 0.8067,E2 233.7112} C_DIS
LIN {X -121.1528,Y -74.2202,Z 191,A -138.4204,B 0.9282,C 0.1522,E1 0.8097,E2 231.6689} C_DIS
LIN {X -119.096,Y -77.4777,Z 191,A -137.148,B 0.9277,C 0.1555,E1 0.8116,E2 230.4381} C_DIS
LIN {X -117.0924,Y -80.4737,Z 191,A -135.3766,B 0.9271,C 0.1586,E1 0.8144,E2 228.6204} C_DIS
LIN {X -115.1486,Y -83.2315,Z 191,A -133.5215,B 0.9267,C 0.1614,E1 0.8176,E2 226.6926} C_DIS
LIN {X -112.9594,Y -86.179,Z 191,A -132.1344,B 0.9261,C 0.1643,E1 0.8199,E2 225.3197} C_DIS
LIN {X -110.1926,Y -89.69,Z 191,A -130.1669,B 0.9255,C 0.1678,E1 0.8234,E2 223.328} C_DIS
LIN {X -108.1068,Y -92.1933,Z 191,A -128.6081,B 0.9251,C 0.1702,E1 0.8263,E2 221.733} C_DIS
LIN {X -104.925,Y -95.7997,Z 191,A -126.4752,B 0.9245,C 0.1736,E1 0.8304,E2 219.5716} C_DIS
LIN {X -101.7366,Y -99.179,Z 191,A -124.2522,B 0.9239,C 0.1767,E1 0.8349,E2 217.2965} C_DIS
LIN {X -98.168,Y -102.7116,Z 191,A -122.2943,B 0.9232,C 0.18,E1 0.8388,E2 215.3488} C_DIS
LIN {X -95.0881,Y -105.5701,Z 191,A -120.3456,B 0.9227,C 0.1825,E1 0.8429,E2 213.3621} C_DIS
LIN {X -92.0402,Y -108.2369,Z 191,A -118.5883,B 0.9223,C 0.1849,E1 0.8467,E2 211.5861} C_DIS
LIN {X -88.4549,Y -111.1862,Z 191,A -116.5599,B 0.9218,C 0.1874,E1 0.8512,E2 209.5341} C_DIS
LIN {X -85.9092,Y -113.1654,Z 191,A -115.0653,B 0.9214,C 0.1889,E1 0.8547,E2 208.0102} C_DIS
LIN {X -81.913,Y -116.09,Z 191,A -112.9854,B 0.9209,C 0.1914,E1 0.8594,E2 205.9175} C_DIS
LIN {X -77.8996,Y -118.8207,Z 191,A -110.9538,B 0.9205,C 0.1935,E1 0.8642,E2 203.8745} C_DIS
LIN {X -74.2093,Y -121.1595,Z 191,A -109.0562,B 0.9201,C 0.1953,E1 0.8689,E2 201.9561} C_DIS
LIN {X -70.2137,Y -123.5181,Z 191,A -107.0713,B 0.9198,C 0.197,E1 0.8738,E2 199.9536} C_DIS
LIN {X -66.4394,Y -125.5868,Z 191,A -105.3019,B 0.9194,C 0.1985,E1 0.8782,E2 198.1788} C_DIS
LIN {X -63.1252,Y -127.2845,Z 191,A -103.7851,B 0.9192,C 0.1997,E1 0.882,E2 196.6593} C_DIS
LIN {X -60.2271,Y -128.6825,Z 191,A -102.334,B 0.919,C 0.2004,E1 0.8858,E2 195.1846} C_DIS
LIN {X -57.3805,Y -129.977,Z 191,A -101.1078,B 0.9188,C 0.2014,E1 0.8889,E2 193.9635} C_DIS
LIN {X -53.6978,Y -131.5409,Z 191,A -99.3538,B 0.9186,C 0.2021,E1 0.8936,E2 192.1875} C_DIS
LIN {X -50.4138,Y -132.8342,Z 191,A -97.9048,B 0.9185,C 0.2029,E1 0.8974,E2 190.7342} C_DIS
LIN {X -47.4353,Y -133.9277,Z 191,A -96.3278,B 0.9185,C 0.2029,E1 0.9018,E2 189.1114} C_DIS
Enddeposition()
END
